Yaskawa INFORM job: A_ROOF_SIDE_0617_2_PAINT_15.JBI

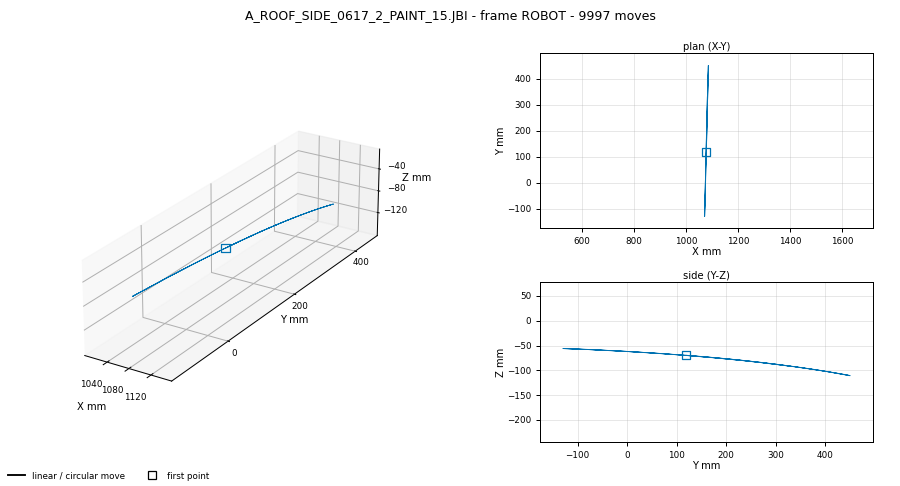
[picture p0: tool path of A_ROOF_SIDE_0617_2_PAINT_15.JBI in frame ROBOT, 9997 of 9997 moves have a stored position in this frame; points joined in program order, loops and branches not executed]
/JOB
//NAME A_ROOF_SIDE_0617_2_PAINT15
//POS
///NPOS 9997,0,0,0,0,0
///TOOL 1
///USER 0
///POSTYPE ROBOT
///RECTAN
///RCONF 1,0,0,0,0,0,0,0,0,0,0,0,0,0,0,0,0,0,0,0,0,0,0,0
C00000=1077.480,118.729,-69.527,173.974,23.685,154.115
C00001=1077.485,118.978,-69.546,173.976,23.687,154.116
C00002=1077.491,119.227,-69.566,173.978,23.689,154.116
C00003=1077.497,119.476,-69.585,173.979,23.692,154.116
C00004=1077.502,119.725,-69.604,173.982,23.695,154.116
C00005=1077.508,119.975,-69.623,173.983,23.697,154.117
C00006=1077.514,120.224,-69.643,173.984,23.699,154.117
C00007=1077.520,120.473,-69.663,173.987,23.702,154.117
C00008=1077.525,120.722,-69.682,173.988,23.704,154.117
C00009=1077.531,120.971,-69.702,173.990,23.707,154.118
C00010=1077.537,121.220,-69.721,173.991,23.709,154.118
C00011=1077.542,121.470,-69.740,173.994,23.711,154.118
C00012=1077.547,121.719,-69.761,173.995,23.714,154.118
C00013=1077.553,121.968,-69.780,173.997,23.716,154.119
C00014=1077.559,122.218,-69.799,173.999,23.719,154.119
C00015=1077.565,122.466,-69.819,174.001,23.721,154.119
C00016=1077.570,122.715,-69.838,174.002,23.723,154.119
C00017=1077.576,122.965,-69.857,174.004,23.726,154.120
C00018=1077.582,123.213,-69.877,174.006,23.728,154.120
C00019=1077.587,123.463,-69.896,174.007,23.730,154.120
C00020=1077.593,123.712,-69.916,174.010,23.733,154.120
C00021=1077.598,123.961,-69.936,174.011,23.735,154.121
C00022=1077.604,124.211,-69.955,174.013,23.738,154.121
C00023=1077.610,124.460,-69.975,174.015,23.740,154.121
C00024=1077.616,124.709,-69.995,174.017,23.743,154.121
C00025=1077.622,124.958,-70.015,174.018,23.745,154.122
C00026=1077.627,125.207,-70.034,174.021,23.747,154.122
C00027=1077.633,125.456,-70.054,174.022,23.750,154.122
C00028=1077.638,125.706,-70.074,174.024,23.752,154.122
C00029=1077.644,125.955,-70.094,174.026,23.754,154.123
C00030=1077.650,126.204,-70.113,174.028,23.757,154.123
C00031=1077.656,126.453,-70.133,174.029,23.759,154.123
C00032=1077.662,126.702,-70.152,174.031,23.761,154.123
C00033=1077.668,126.983,-70.174,174.033,23.764,154.124
C00034=1077.674,127.265,-70.197,174.035,23.767,154.124
C00035=1077.681,127.545,-70.219,174.037,23.769,154.124
C00036=1077.687,127.826,-70.242,174.039,23.772,154.124
C00037=1077.693,128.075,-70.261,174.041,23.775,154.125
C00038=1077.699,128.324,-70.281,174.043,23.777,154.125
C00039=1077.704,128.574,-70.301,174.045,23.779,154.125
C00040=1077.710,128.823,-70.321,174.047,23.782,154.125
C00041=1077.716,129.072,-70.340,174.048,23.784,154.125
C00042=1077.722,129.321,-70.360,174.050,23.786,154.126
C00043=1077.728,129.570,-70.380,174.052,23.789,154.126
C00044=1077.733,129.819,-70.400,174.054,23.791,154.126
C00045=1077.739,130.068,-70.420,174.056,23.793,154.126
C00046=1077.745,130.317,-70.439,174.058,23.796,154.127
C00047=1077.750,130.567,-70.459,174.059,23.798,154.127
C00048=1077.756,130.815,-70.479,174.062,23.800,154.127
C00049=1077.762,131.065,-70.500,174.063,23.803,154.127
C00050=1077.768,131.315,-70.519,174.065,23.805,154.128
C00051=1077.774,131.563,-70.539,174.067,23.807,154.128
C00052=1077.780,131.812,-70.559,174.069,23.810,154.128
C00053=1077.785,132.062,-70.579,174.070,23.812,154.128
C00054=1077.791,132.311,-70.599,174.073,23.814,154.128
C00055=1077.797,132.560,-70.619,174.074,23.817,154.129
C00056=1077.802,132.809,-70.639,174.076,23.819,154.129
C00057=1077.808,133.058,-70.658,174.078,23.821,154.129
C00058=1077.813,133.307,-70.679,174.080,23.824,154.129
C00059=1077.819,133.556,-70.699,174.081,23.826,154.130
C00060=1077.824,133.805,-70.719,174.084,23.829,154.130
C00061=1077.830,134.055,-70.739,174.085,23.831,154.130
C00062=1077.835,134.304,-70.759,174.087,23.833,154.130
C00063=1077.841,134.553,-70.779,174.089,23.836,154.131
C00064=1077.846,134.802,-70.800,174.091,23.838,154.131
C00065=1077.853,135.051,-70.820,174.092,23.840,154.131
C00066=1077.859,135.300,-70.840,174.095,23.843,154.131
C00067=1077.864,135.550,-70.860,174.096,23.845,154.132
C00068=1077.870,135.799,-70.880,174.098,23.848,154.132
C00069=1077.875,136.048,-70.900,174.100,23.850,154.132
C00070=1077.881,136.297,-70.920,174.102,23.853,154.132
C00071=1077.886,136.546,-70.941,174.103,23.854,154.132
C00072=1077.892,136.794,-70.961,174.106,23.857,154.133
C00073=1077.898,137.044,-70.981,174.108,23.859,154.133
C00074=1077.904,137.293,-71.002,174.109,23.862,154.133
C00075=1077.910,137.542,-71.022,174.112,23.864,154.133
C00076=1077.915,137.792,-71.041,174.113,23.866,154.133
C00077=1077.920,138.041,-71.062,174.115,23.869,154.134
C00078=1077.926,138.290,-71.082,174.117,23.871,154.134
C00079=1077.932,138.539,-71.103,174.119,23.874,154.134
C00080=1077.937,138.788,-71.123,174.120,23.876,154.134
C00081=1077.944,139.037,-71.143,174.123,23.878,154.135
C00082=1077.949,139.286,-71.164,174.124,23.881,154.135
C00083=1077.955,139.535,-71.184,174.126,23.883,154.135
C00084=1077.960,139.784,-71.204,174.128,23.885,154.135
C00085=1077.966,140.033,-71.224,174.130,23.888,154.136
C00086=1077.971,140.282,-71.245,174.132,23.890,154.136
C00087=1077.977,140.532,-71.266,174.134,23.892,154.136
C00088=1077.983,140.781,-71.286,174.136,23.895,154.136
C00089=1077.988,141.030,-71.306,174.137,23.897,154.136
C00090=1077.994,141.279,-71.327,174.140,23.900,154.137
C00091=1078.000,141.527,-71.348,174.141,23.902,154.137
C00092=1078.005,141.777,-71.368,174.143,23.904,154.137
C00093=1078.010,142.026,-71.389,174.145,23.907,154.137
C00094=1078.016,142.276,-71.410,174.147,23.909,154.138
C00095=1078.022,142.524,-71.430,174.149,23.912,154.138
C00096=1078.028,142.773,-71.450,174.151,23.913,154.138
C00097=1078.034,143.054,-71.473,174.153,23.916,154.138
C00098=1078.040,143.335,-71.497,174.155,23.919,154.139
C00099=1078.047,143.616,-71.520,174.158,23.922,154.139
C00100=1078.053,143.897,-71.543,174.160,23.924,154.139
C00101=1078.058,144.146,-71.563,174.161,23.927,154.139
C00102=1078.064,144.395,-71.585,174.164,23.929,154.139
C00103=1078.071,144.644,-71.605,174.166,23.932,154.140
C00104=1078.076,144.893,-71.625,174.167,23.933,154.140
C00105=1078.081,145.143,-71.646,174.170,23.936,154.140
C00106=1078.086,145.392,-71.667,174.171,23.938,154.140
C00107=1078.093,145.641,-71.688,174.173,23.941,154.141
C00108=1078.098,145.890,-71.708,174.175,23.943,154.141
C00109=1078.104,146.139,-71.729,174.177,23.945,154.141
C00110=1078.109,146.388,-71.749,174.179,23.948,154.141
C00111=1078.116,146.637,-71.770,174.181,23.950,154.141
C00112=1078.121,146.886,-71.791,174.183,23.953,154.142
C00113=1078.126,147.135,-71.811,174.185,23.954,154.142
C00114=1078.133,147.384,-71.833,174.187,23.957,154.142
C00115=1078.138,147.633,-71.854,174.189,23.959,154.142
C00116=1078.144,147.882,-71.874,174.190,23.962,154.143
C00117=1078.149,148.131,-71.894,174.193,23.964,154.143
C00118=1078.155,148.381,-71.916,174.194,23.966,154.143
C00119=1078.160,148.630,-71.936,174.196,23.969,154.143
C00120=1078.166,148.878,-71.958,174.199,23.971,154.143
C00121=1078.172,149.128,-71.979,174.200,23.973,154.144
C00122=1078.177,149.377,-71.999,174.203,23.976,154.144
C00123=1078.183,149.625,-72.020,174.204,23.978,154.144
C00124=1078.189,149.874,-72.040,174.206,23.981,154.144
C00125=1078.195,150.124,-72.061,174.209,23.983,154.145
C00126=1078.200,150.373,-72.082,174.210,23.985,154.145
C00127=1078.205,150.622,-72.103,174.212,23.987,154.145
C00128=1078.212,150.871,-72.125,174.214,23.990,154.145
C00129=1078.217,151.120,-72.145,174.216,23.992,154.145
C00130=1078.222,151.369,-72.166,174.218,23.995,154.146
C00131=1078.228,151.619,-72.187,174.220,23.997,154.146
C00132=1078.234,151.867,-72.209,174.222,23.999,154.146
C00133=1078.239,152.116,-72.229,174.224,24.002,154.146
C00134=1078.245,152.365,-72.251,174.226,24.004,154.147
C00135=1078.250,152.614,-72.271,174.228,24.007,154.147
C00136=1078.256,152.863,-72.293,174.230,24.008,154.147
C00137=1078.262,153.113,-72.314,174.232,24.011,154.147
C00138=1078.267,153.361,-72.335,174.234,24.013,154.147
C00139=1078.273,153.610,-72.355,174.236,24.016,154.148
C00140=1078.279,153.860,-72.377,174.238,24.018,154.148
C00141=1078.284,154.109,-72.398,174.240,24.021,154.148
C00142=1078.290,154.358,-72.419,174.242,24.022,154.148
C00143=1078.296,154.607,-72.440,174.244,24.025,154.149
C00144=1078.301,154.856,-72.461,174.245,24.027,154.149
C00145=1078.307,155.105,-72.483,174.248,24.030,154.149
C00146=1078.312,155.354,-72.503,174.250,24.032,154.149
C00147=1078.319,155.603,-72.525,174.251,24.034,154.149
C00148=1078.324,155.852,-72.546,174.254,24.036,154.150
C00149=1078.329,156.101,-72.567,174.256,24.039,154.150
C00150=1078.335,156.350,-72.589,174.257,24.041,154.150
C00151=1078.340,156.599,-72.610,174.260,24.044,154.150
C00152=1078.346,156.848,-72.631,174.262,24.046,154.150
C00153=1078.352,157.097,-72.652,174.264,24.048,154.151
C00154=1078.357,157.346,-72.674,174.266,24.051,154.151
C00155=1078.363,157.595,-72.695,174.268,24.053,154.151
C00156=1078.368,157.844,-72.716,174.270,24.055,154.151
C00157=1078.374,158.093,-72.738,174.272,24.058,154.151
C00158=1078.380,158.343,-72.759,174.274,24.060,154.152
C00159=1078.385,158.591,-72.780,174.276,24.062,154.152
C00160=1078.391,158.840,-72.802,174.278,24.065,154.152
C00161=1078.398,159.121,-72.825,174.280,24.068,154.152
C00162=1078.404,159.402,-72.850,174.283,24.070,154.153
C00163=1078.410,159.682,-72.874,174.285,24.072,154.153
C00164=1078.417,159.963,-72.898,174.287,24.075,154.153
C00165=1078.422,160.212,-72.919,174.290,24.077,154.153
C00166=1078.427,160.461,-72.941,174.291,24.080,154.154
C00167=1078.433,160.710,-72.963,174.293,24.082,154.154
C00168=1078.439,160.959,-72.983,174.296,24.085,154.154
C00169=1078.445,161.208,-73.005,174.297,24.086,154.154
C00170=1078.450,161.457,-73.026,174.299,24.089,154.154
C00171=1078.456,161.706,-73.048,174.302,24.091,154.155
C00172=1078.461,161.955,-73.070,174.303,24.094,154.155
C00173=1078.467,162.204,-73.092,174.305,24.096,154.155
C00174=1078.472,162.453,-73.113,174.308,24.099,154.155
C00175=1078.478,162.702,-73.135,174.310,24.101,154.155
C00176=1078.483,162.951,-73.157,174.311,24.104,154.156
C00177=1078.488,163.200,-73.178,174.314,24.106,154.156
C00178=1078.494,163.449,-73.199,174.316,24.109,154.156
C00179=1078.499,163.698,-73.221,174.317,24.111,154.156
C00180=1078.505,163.947,-73.243,174.320,24.113,154.157
C00181=1078.510,164.196,-73.265,174.322,24.116,154.157
C00182=1078.516,164.446,-73.286,174.324,24.118,154.157
C00183=1078.521,164.694,-73.308,174.326,24.120,154.157
C00184=1078.527,164.944,-73.330,174.328,24.123,154.158
C00185=1078.532,165.192,-73.352,174.330,24.125,154.158
C00186=1078.538,165.442,-73.373,174.332,24.128,154.158
C00187=1078.543,165.690,-73.395,174.334,24.130,154.158
C00188=1078.549,165.940,-73.417,174.336,24.132,154.158
C00189=1078.554,166.188,-73.439,174.338,24.134,154.159
C00190=1078.560,166.437,-73.461,174.340,24.137,154.159
C00191=1078.565,166.686,-73.483,174.343,24.140,154.159
C00192=1078.571,166.935,-73.505,174.345,24.142,154.159
C00193=1078.576,167.184,-73.526,174.346,24.144,154.160
C00194=1078.582,167.433,-73.548,174.349,24.146,154.160
C00195=1078.587,167.682,-73.570,174.351,24.149,154.160
C00196=1078.592,167.931,-73.592,174.352,24.151,154.160
C00197=1078.598,168.180,-73.613,174.355,24.154,154.160
C00198=1078.603,168.429,-73.636,174.357,24.156,154.161
C00199=1078.609,168.677,-73.658,174.359,24.159,154.161
C00200=1078.615,168.927,-73.680,174.361,24.161,154.161
C00201=1078.620,169.175,-73.701,174.363,24.163,154.161
C00202=1078.626,169.425,-73.723,174.365,24.166,154.161
C00203=1078.632,169.674,-73.745,174.368,24.168,154.162
C00204=1078.637,169.923,-73.767,174.369,24.170,154.162
C00205=1078.642,170.172,-73.790,174.372,24.172,154.162
C00206=1078.648,170.420,-73.811,174.374,24.175,154.162
C00207=1078.653,170.670,-73.833,174.376,24.177,154.162
C00208=1078.660,170.919,-73.855,174.378,24.180,154.163
C00209=1078.665,171.167,-73.878,174.380,24.182,154.163
C00210=1078.670,171.417,-73.900,174.382,24.185,154.163
C00211=1078.676,171.665,-73.921,174.385,24.187,154.163
C00212=1078.681,171.915,-73.943,174.386,24.189,154.164
C00213=1078.688,172.163,-73.966,174.388,24.191,154.164
C00214=1078.692,172.412,-73.987,174.391,24.194,154.164
C00215=1078.698,172.662,-74.010,174.393,24.196,154.164
C00216=1078.704,172.910,-74.032,174.395,24.199,154.164
C00217=1078.709,173.159,-74.054,174.397,24.201,154.165
C00218=1078.715,173.409,-74.076,174.399,24.203,154.165
C00219=1078.721,173.657,-74.099,174.402,24.206,154.165
C00220=1078.726,173.906,-74.120,174.403,24.208,154.165
C00221=1078.732,174.155,-74.142,174.405,24.210,154.165
C00222=1078.738,174.404,-74.165,174.408,24.212,154.166
C00223=1078.743,174.653,-74.187,174.410,24.215,154.166
C00224=1078.749,174.901,-74.209,174.412,24.217,154.166
C00225=1078.755,175.182,-74.235,174.415,24.220,154.166
C00226=1078.761,175.462,-74.260,174.417,24.223,154.166
C00227=1078.768,175.743,-74.284,174.419,24.225,154.167
C00228=1078.774,176.023,-74.309,174.422,24.227,154.167
C00229=1078.780,176.272,-74.332,174.424,24.230,154.167
C00230=1078.785,176.522,-74.354,174.426,24.232,154.167
C00231=1078.791,176.770,-74.376,174.428,24.235,154.168
C00232=1078.796,177.019,-74.398,174.430,24.237,154.168
C00233=1078.802,177.268,-74.421,174.433,24.239,154.168
C00234=1078.809,177.517,-74.443,174.435,24.242,154.168
C00235=1078.813,177.765,-74.465,174.437,24.244,154.168
C00236=1078.819,178.014,-74.488,174.439,24.246,154.169
C00237=1078.825,178.263,-74.510,174.441,24.248,154.169
C00238=1078.831,178.512,-74.533,174.443,24.251,154.169
C00239=1078.837,178.762,-74.555,174.446,24.253,154.169
C00240=1078.842,179.010,-74.578,174.448,24.255,154.169
C00241=1078.848,179.259,-74.599,174.450,24.258,154.170
C00242=1078.854,179.508,-74.622,174.452,24.260,154.170
C00243=1078.859,179.757,-74.645,174.454,24.262,154.170
C00244=1078.865,180.006,-74.667,174.457,24.265,154.170
C00245=1078.871,180.254,-74.689,174.459,24.267,154.170
C00246=1078.876,180.503,-74.712,174.461,24.270,154.171
C00247=1078.882,180.753,-74.735,174.463,24.272,154.171
C00248=1078.888,181.001,-74.757,174.465,24.274,154.171
C00249=1078.894,181.250,-74.780,174.467,24.276,154.171
C00250=1078.899,181.500,-74.802,174.470,24.279,154.171
C00251=1078.905,181.749,-74.825,174.472,24.281,154.171
C00252=1078.911,181.997,-74.847,174.475,24.283,154.172
C00253=1078.916,182.246,-74.869,174.476,24.285,154.172
C00254=1078.922,182.495,-74.892,174.479,24.287,154.172
C00255=1078.928,182.744,-74.915,174.481,24.290,154.172
C00256=1078.934,182.993,-74.938,174.483,24.292,154.172
C00257=1078.940,183.242,-74.960,174.486,24.294,154.173
C00258=1078.945,183.491,-74.983,174.488,24.297,154.173
C00259=1078.951,183.740,-75.006,174.490,24.299,154.173
C00260=1078.957,183.989,-75.029,174.492,24.301,154.173
C00261=1078.963,184.238,-75.050,174.494,24.304,154.173
C00262=1078.968,184.486,-75.073,174.497,24.306,154.173
C00263=1078.974,184.735,-75.096,174.499,24.308,154.174
C00264=1078.980,184.984,-75.119,174.501,24.311,154.174
C00265=1078.985,185.233,-75.142,174.504,24.313,154.174
C00266=1078.991,185.482,-75.165,174.506,24.316,154.174
C00267=1078.997,185.731,-75.187,174.507,24.318,154.174
C00268=1079.002,185.980,-75.210,174.510,24.320,154.175
C00269=1079.007,186.229,-75.233,174.512,24.323,154.175
C00270=1079.012,186.478,-75.256,174.514,24.325,154.175
C00271=1079.018,186.726,-75.279,174.517,24.328,154.175
C00272=1079.024,186.975,-75.302,174.519,24.330,154.176
C00273=1079.030,187.224,-75.325,174.521,24.333,154.176
C00274=1079.035,187.473,-75.348,174.523,24.334,154.176
C00275=1079.040,187.722,-75.371,174.525,24.337,154.176
C00276=1079.045,187.971,-75.394,174.527,24.340,154.177
C00277=1079.051,188.219,-75.417,174.530,24.342,154.177
C00278=1079.057,188.468,-75.440,174.532,24.345,154.177
C00279=1079.062,188.718,-75.463,174.535,24.347,154.177
C00280=1079.068,188.966,-75.486,174.537,24.350,154.177
C00281=1079.073,189.215,-75.509,174.539,24.352,154.177
C00282=1079.079,189.464,-75.532,174.542,24.354,154.178
C00283=1079.084,189.712,-75.555,174.543,24.356,154.178
C00284=1079.089,189.962,-75.578,174.545,24.359,154.178
C00285=1079.095,190.211,-75.601,174.548,24.361,154.178
C00286=1079.101,190.459,-75.624,174.550,24.364,154.179
C00287=1079.106,190.708,-75.647,174.553,24.366,154.179
C00288=1079.111,190.958,-75.671,174.555,24.369,154.179
C00289=1079.118,191.238,-75.697,174.557,24.371,154.179
C00290=1079.124,191.517,-75.722,174.560,24.374,154.180
C00291=1079.131,191.797,-75.749,174.563,24.377,154.180
C00292=1079.136,192.077,-75.775,174.565,24.379,154.180
C00293=1079.142,192.326,-75.798,174.567,24.382,154.180
C00294=1079.148,192.575,-75.821,174.570,24.384,154.180
C00295=1079.153,192.824,-75.844,174.572,24.387,154.181
C00296=1079.159,193.072,-75.868,174.574,24.389,154.181
C00297=1079.165,193.321,-75.891,174.577,24.392,154.181
C00298=1079.170,193.570,-75.914,174.579,24.394,154.181
C00299=1079.175,193.819,-75.937,174.581,24.396,154.181
C00300=1079.181,194.068,-75.960,174.583,24.398,154.182
C00301=1079.187,194.316,-75.984,174.585,24.401,154.182
C00302=1079.192,194.566,-76.008,174.588,24.403,154.182
C00303=1079.198,194.814,-76.031,174.590,24.406,154.182
C00304=1079.204,195.063,-76.054,174.592,24.408,154.182
C00305=1079.210,195.312,-76.077,174.595,24.411,154.183
C00306=1079.215,195.561,-76.101,174.597,24.413,154.183
C00307=1079.221,195.810,-76.124,174.599,24.416,154.183
C00308=1079.227,196.059,-76.148,174.602,24.418,154.183
C00309=1079.232,196.308,-76.171,174.604,24.420,154.184
C00310=1079.238,196.557,-76.194,174.606,24.423,154.184
C00311=1079.244,196.805,-76.218,174.609,24.425,154.184
C00312=1079.249,197.054,-76.241,174.611,24.427,154.184
C00313=1079.255,197.303,-76.264,174.614,24.430,154.184
C00314=1079.261,197.552,-76.288,174.616,24.432,154.184
C00315=1079.266,197.801,-76.312,174.618,24.434,154.185
C00316=1079.272,198.049,-76.335,174.621,24.437,154.185
C00317=1079.277,198.298,-76.358,174.623,24.439,154.185
C00318=1079.283,198.547,-76.383,174.625,24.442,154.185
C00319=1079.289,198.796,-76.406,174.628,24.444,154.185
C00320=1079.294,199.045,-76.429,174.630,24.447,154.186
C00321=1079.300,199.294,-76.453,174.632,24.449,154.186
C00322=1079.306,199.542,-76.476,174.635,24.451,154.186
C00323=1079.311,199.791,-76.500,174.637,24.454,154.186
C00324=1079.317,200.040,-76.523,174.640,24.456,154.186
C00325=1079.323,200.289,-76.547,174.642,24.459,154.187
C00326=1079.328,200.538,-76.571,174.643,24.460,154.187
C00327=1079.334,200.786,-76.594,174.646,24.463,154.187
C00328=1079.339,201.036,-76.618,174.648,24.465,154.187
C00329=1079.345,201.284,-76.641,174.651,24.467,154.187
C00330=1079.351,201.532,-76.665,174.653,24.470,154.188
C00331=1079.357,201.782,-76.689,174.655,24.472,154.188
C00332=1079.363,202.030,-76.713,174.658,24.475,154.188
C00333=1079.368,202.280,-76.736,174.660,24.477,154.188
C00334=1079.374,202.528,-76.760,174.662,24.480,154.189
C00335=1079.380,202.777,-76.785,174.665,24.482,154.189
C00336=1079.386,203.026,-76.807,174.668,24.485,154.189
C00337=1079.391,203.275,-76.832,174.670,24.487,154.189
C00338=1079.396,203.523,-76.856,174.673,24.490,154.189
C00339=1079.402,203.772,-76.879,174.675,24.492,154.189
C00340=1079.407,204.021,-76.903,174.677,24.495,154.190
C00341=1079.413,204.269,-76.927,174.680,24.497,154.190
C00342=1079.419,204.519,-76.951,174.682,24.499,154.190
C00343=1079.424,204.767,-76.975,174.684,24.502,154.190
C00344=1079.430,205.016,-76.999,174.687,24.504,154.191
C00345=1079.435,205.265,-77.022,174.689,24.507,154.191
C00346=1079.441,205.514,-77.046,174.692,24.509,154.191
C00347=1079.447,205.763,-77.071,174.694,24.512,154.191
C00348=1079.453,206.011,-77.095,174.696,24.514,154.191
C00349=1079.458,206.260,-77.119,174.699,24.517,154.192
C00350=1079.463,206.509,-77.143,174.701,24.519,154.192
C00351=1079.470,206.758,-77.167,174.703,24.521,154.192
C00352=1079.475,207.006,-77.191,174.706,24.524,154.192
C00353=1079.498,208.041,-77.291,174.808,24.578,154.191
C00354=1079.507,208.442,-77.330,174.812,24.584,154.192
C00355=1079.516,208.843,-77.371,174.815,24.589,154.192
C00356=1079.526,209.243,-77.410,174.819,24.595,154.193
C00357=1079.535,209.644,-77.449,174.823,24.601,154.194
C00358=1079.541,209.893,-77.474,174.825,24.604,154.194
C00359=1079.546,210.141,-77.499,174.827,24.607,154.194
C00360=1079.552,210.391,-77.523,174.829,24.611,154.195
C00361=1079.558,210.639,-77.548,174.832,24.614,154.195
C00362=1079.564,210.888,-77.573,174.834,24.617,154.196
C00363=1079.569,211.137,-77.597,174.837,24.621,154.196
C00364=1079.575,211.385,-77.622,174.839,24.625,154.197
C00365=1079.580,211.634,-77.647,174.841,24.628,154.197
C00366=1079.586,211.883,-77.673,174.843,24.631,154.198
C00367=1079.592,212.132,-77.697,174.845,24.635,154.198
C00368=1079.598,212.380,-77.722,174.848,24.638,154.198
C00369=1079.603,212.629,-77.747,174.850,24.641,154.199
C00370=1079.609,212.877,-77.772,174.853,24.645,154.199
C00371=1079.615,213.127,-77.796,174.855,24.648,154.200
C00372=1079.621,213.375,-77.821,174.857,24.651,154.200
C00373=1079.626,213.624,-77.846,174.860,24.655,154.201
C00374=1079.631,213.872,-77.872,174.862,24.659,154.201
C00375=1079.637,214.121,-77.896,174.864,24.662,154.201
C00376=1079.643,214.369,-77.921,174.866,24.665,154.202
C00377=1079.649,214.619,-77.946,174.868,24.669,154.202
C00378=1079.654,214.868,-77.972,174.871,24.672,154.203
C00379=1079.659,215.116,-77.996,174.873,24.675,154.203
C00380=1079.666,215.365,-78.021,174.875,24.679,154.204
C00381=1079.671,215.613,-78.046,174.877,24.682,154.204
C00382=1079.677,215.862,-78.071,174.880,24.686,154.204
C00383=1079.683,216.111,-78.097,174.882,24.690,154.205
C00384=1079.688,216.359,-78.122,174.885,24.693,154.205
C00385=1079.694,216.608,-78.146,174.887,24.696,154.206
C00386=1079.700,216.856,-78.171,174.889,24.699,154.206
C00387=1079.705,217.105,-78.197,174.892,24.703,154.207
C00388=1079.711,217.355,-78.222,174.894,24.706,154.207
C00389=1079.717,217.603,-78.247,174.896,24.710,154.208
C00390=1079.722,217.852,-78.273,174.898,24.713,154.208
C00391=1079.728,218.101,-78.297,174.900,24.716,154.208
C00392=1079.734,218.349,-78.322,174.903,24.720,154.209
C00393=1079.740,218.598,-78.348,174.906,24.723,154.209
C00394=1079.745,218.847,-78.374,174.908,24.727,154.210
C00395=1079.751,219.094,-78.399,174.910,24.730,154.210
C00396=1079.757,219.344,-78.423,174.913,24.734,154.211
C00397=1079.762,219.593,-78.449,174.915,24.737,154.211
C00398=1079.768,219.841,-78.474,174.917,24.740,154.211
C00399=1079.774,220.089,-78.500,174.919,24.744,154.212
C00400=1079.780,220.338,-78.525,174.922,24.747,154.212
C00401=1079.785,220.586,-78.550,174.924,24.750,154.213
C00402=1079.791,220.836,-78.575,174.926,24.754,154.213
C00403=1079.797,221.085,-78.601,174.929,24.757,154.214
C00404=1079.803,221.333,-78.626,174.932,24.761,154.214
C00405=1079.808,221.581,-78.651,174.934,24.764,154.214
C00406=1079.817,221.987,-78.693,174.937,24.769,154.215
C00407=1079.827,222.391,-78.735,174.941,24.775,154.216
C00408=1079.835,222.797,-78.776,174.945,24.781,154.216
C00409=1079.845,223.201,-78.818,174.949,24.786,154.217
C00410=1079.851,223.450,-78.844,174.951,24.790,154.218
C00411=1079.857,223.699,-78.869,174.953,24.793,154.218
C00412=1079.863,223.948,-78.895,174.956,24.797,154.218
C00413=1079.867,224.196,-78.920,174.958,24.800,154.219
C00414=1079.874,224.445,-78.946,174.960,24.803,154.219
C00415=1079.879,224.694,-78.972,174.963,24.807,154.220
C00416=1079.885,224.942,-78.997,174.965,24.811,154.220
C00417=1079.890,225.190,-79.023,174.968,24.814,154.221
C00418=1079.896,225.439,-79.048,174.970,24.817,154.221
C00419=1079.902,225.688,-79.074,174.973,24.820,154.222
C00420=1079.907,225.937,-79.100,174.975,24.824,154.222
C00421=1079.914,226.185,-79.126,174.977,24.827,154.222
C00422=1079.919,226.433,-79.151,174.979,24.830,154.223
C00423=1079.925,226.682,-79.177,174.982,24.835,154.223
C00424=1079.930,226.931,-79.203,174.984,24.838,154.224
C00425=1079.937,227.180,-79.228,174.987,24.841,154.224
C00426=1079.942,227.428,-79.255,174.990,24.844,154.225
C00427=1079.948,227.677,-79.281,174.992,24.848,154.225
C00428=1079.954,227.926,-79.306,174.994,24.851,154.225
C00429=1079.959,228.174,-79.331,174.996,24.854,154.226
C00430=1079.964,228.423,-79.357,174.999,24.858,154.226
C00431=1079.971,228.671,-79.383,175.001,24.862,154.227
C00432=1079.976,228.920,-79.409,175.003,24.865,154.227
C00433=1079.983,229.169,-79.435,175.006,24.868,154.228
C00434=1079.988,229.417,-79.461,175.009,24.871,154.228
C00435=1079.994,229.666,-79.487,175.011,24.875,154.228
C00436=1080.000,229.915,-79.513,175.014,24.879,154.229
C00437=1080.006,230.163,-79.539,175.016,24.882,154.229
C00438=1080.011,230.411,-79.565,175.018,24.885,154.230
C00439=1080.016,230.660,-79.591,175.020,24.889,154.230
C00440=1080.023,230.908,-79.617,175.023,24.892,154.231
C00441=1080.028,231.157,-79.643,175.025,24.895,154.231
C00442=1080.034,231.406,-79.669,175.027,24.899,154.231
C00443=1080.039,231.655,-79.695,175.030,24.903,154.232
C00444=1080.045,231.904,-79.721,175.033,24.906,154.232
C00445=1080.051,232.152,-79.747,175.035,24.909,154.233
C00446=1080.057,232.401,-79.773,175.038,24.913,154.233
C00447=1080.063,232.649,-79.800,175.040,24.916,154.234
C00448=1080.068,232.898,-79.826,175.042,24.919,154.234
C00449=1080.073,233.146,-79.852,175.045,24.923,154.235
C00450=1080.079,233.395,-79.878,175.047,24.926,154.235
C00451=1080.084,233.643,-79.905,175.049,24.930,154.235
C00452=1080.091,233.892,-79.930,175.053,24.933,154.236
C00453=1080.096,234.140,-79.957,175.055,24.937,154.236
C00454=1080.102,234.389,-79.983,175.057,24.940,154.237
C00455=1080.108,234.637,-80.009,175.060,24.943,154.237
C00456=1080.113,234.886,-80.036,175.062,24.947,154.238
C00457=1080.119,235.135,-80.062,175.064,24.950,154.238
C00458=1080.128,235.531,-80.104,175.069,24.956,154.239
C00459=1080.137,235.928,-80.146,175.072,24.961,154.239
C00460=1080.146,236.324,-80.188,175.076,24.967,154.240
C00461=1080.155,236.720,-80.230,175.080,24.973,154.241
C00462=1080.161,236.969,-80.256,175.082,24.976,154.241
C00463=1080.166,237.218,-80.283,175.085,24.979,154.242
C00464=1080.173,237.467,-80.310,175.088,24.983,154.242
C00465=1080.178,237.716,-80.336,175.090,24.986,154.243
C00466=1080.184,237.964,-80.363,175.092,24.989,154.243
C00467=1080.190,238.212,-80.389,175.095,24.993,154.243
C00468=1080.196,238.461,-80.416,175.097,24.996,154.244
C00469=1080.201,238.710,-80.442,175.099,25.000,154.244
C00470=1080.207,238.958,-80.469,175.102,25.003,154.245
C00471=1080.213,239.206,-80.495,175.104,25.007,154.245
C00472=1080.218,239.455,-80.522,175.107,25.010,154.246
C00473=1080.224,239.703,-80.548,175.110,25.013,154.246
C00474=1080.229,239.952,-80.576,175.112,25.017,154.246
C00475=1080.235,240.201,-80.602,175.115,25.021,154.247
C00476=1080.240,240.449,-80.628,175.117,25.024,154.247
C00477=1080.246,240.697,-80.655,175.119,25.027,154.248
C00478=1080.253,240.946,-80.682,175.122,25.031,154.248
C00479=1080.258,241.195,-80.709,175.124,25.034,154.249
C00480=1080.264,241.443,-80.735,175.127,25.037,154.249
C00481=1080.270,241.692,-80.762,175.130,25.041,154.250
C00482=1080.276,241.940,-80.789,175.132,25.044,154.250
C00483=1080.281,242.188,-80.815,175.135,25.048,154.250
C00484=1080.287,242.437,-80.842,175.137,25.051,154.251
C00485=1080.293,242.686,-80.869,175.139,25.055,154.251
C00486=1080.299,242.934,-80.896,175.142,25.058,154.252
C00487=1080.304,243.183,-80.923,175.144,25.061,154.252
C00488=1080.310,243.431,-80.949,175.147,25.065,154.253
C00489=1080.315,243.680,-80.977,175.150,25.069,154.253
C00490=1080.321,243.928,-81.003,175.152,25.072,154.253
C00491=1080.327,244.176,-81.030,175.155,25.076,154.254
C00492=1080.332,244.425,-81.057,175.157,25.079,154.254
C00493=1080.338,244.674,-81.084,175.160,25.082,154.255
C00494=1080.344,244.923,-81.111,175.162,25.086,154.255
C00495=1080.349,245.171,-81.139,175.164,25.089,154.256
C00496=1080.355,245.419,-81.165,175.167,25.093,154.256
C00497=1080.361,245.667,-81.192,175.169,25.096,154.257
C00498=1080.367,245.917,-81.220,175.173,25.100,154.257
C00499=1080.372,246.165,-81.246,175.175,25.103,154.257
C00500=1080.378,246.413,-81.273,175.177,25.107,154.258
C00501=1080.383,246.661,-81.301,175.180,25.110,154.258
C00502=1080.389,246.910,-81.328,175.182,25.114,154.259
C00503=1080.396,247.159,-81.355,175.185,25.117,154.259
C00504=1080.401,247.408,-81.382,175.187,25.120,154.260
C00505=1080.407,247.655,-81.409,175.189,25.124,154.260
C00506=1080.412,247.904,-81.436,175.192,25.127,154.260
C00507=1080.417,248.152,-81.463,175.195,25.131,154.261
C00508=1080.423,248.400,-81.491,175.198,25.135,154.261
C00509=1080.429,248.649,-81.518,175.200,25.138,154.262
C00510=1080.437,249.039,-81.561,175.204,25.144,154.263
C00511=1080.445,249.429,-81.604,175.208,25.149,154.263
C00512=1080.455,249.819,-81.647,175.211,25.155,154.264
C00513=1080.463,250.208,-81.690,175.216,25.161,154.265
C00514=1080.470,250.458,-81.717,175.218,25.164,154.265
C00515=1080.475,250.706,-81.745,175.221,25.167,154.266
C00516=1080.481,250.954,-81.771,175.223,25.171,154.266
C00517=1080.486,251.202,-81.799,175.226,25.174,154.266
C00518=1080.492,251.451,-81.827,175.229,25.178,154.267
C00519=1080.498,251.699,-81.854,175.231,25.181,154.267
C00520=1080.503,251.948,-81.881,175.234,25.185,154.268
C00521=1080.510,252.196,-81.909,175.236,25.188,154.268
C00522=1080.515,252.445,-81.936,175.239,25.192,154.269
C00523=1080.520,252.693,-81.964,175.241,25.195,154.269
C00524=1080.526,252.941,-81.991,175.244,25.199,154.270
C00525=1080.532,253.190,-82.019,175.246,25.202,154.270
C00526=1080.538,253.438,-82.047,175.249,25.206,154.271
C00527=1080.543,253.686,-82.074,175.252,25.209,154.271
C00528=1080.549,253.935,-82.102,175.254,25.213,154.271
C00529=1080.555,254.184,-82.129,175.257,25.216,154.272
C00530=1080.560,254.432,-82.157,175.259,25.220,154.272
C00531=1080.566,254.680,-82.185,175.262,25.223,154.273
C00532=1080.572,254.929,-82.212,175.264,25.226,154.273
C00533=1080.578,255.177,-82.240,175.267,25.230,154.274
C00534=1080.583,255.426,-82.268,175.270,25.234,154.274
C00535=1080.589,255.674,-82.295,175.273,25.238,154.275
C00536=1080.595,255.923,-82.323,175.275,25.241,154.275
C00537=1080.600,256.171,-82.351,175.278,25.244,154.275
C00538=1080.607,256.419,-82.379,175.280,25.248,154.276
C00539=1080.612,256.668,-82.406,175.283,25.251,154.276
C00540=1080.617,256.916,-82.434,175.285,25.254,154.277
C00541=1080.624,257.164,-82.462,175.288,25.258,154.277
C00542=1080.629,257.412,-82.490,175.290,25.261,154.278
C00543=1080.635,257.662,-82.517,175.293,25.265,154.278
C00544=1080.641,257.909,-82.545,175.296,25.269,154.279
C00545=1080.647,258.158,-82.573,175.298,25.272,154.279
C00546=1080.652,258.406,-82.601,175.301,25.276,154.280
C00547=1080.658,258.655,-82.629,175.303,25.279,154.280
C00548=1080.664,258.903,-82.657,175.306,25.282,154.280
C00549=1080.670,259.151,-82.685,175.308,25.286,154.281
C00550=1080.675,259.400,-82.713,175.311,25.289,154.281
C00551=1080.682,259.649,-82.740,175.314,25.293,154.282
C00552=1080.687,259.897,-82.768,175.317,25.297,154.282
C00553=1080.693,260.145,-82.796,175.319,25.300,154.283
C00554=1080.698,260.393,-82.824,175.322,25.304,154.283
C00555=1080.705,260.642,-82.852,175.325,25.307,154.283
C00556=1080.710,260.890,-82.880,175.327,25.310,154.284
C00557=1080.716,261.139,-82.908,175.330,25.314,154.284
C00558=1080.722,261.387,-82.936,175.332,25.317,154.285
C00559=1080.728,261.636,-82.964,175.336,25.321,154.285
C00560=1080.734,261.884,-82.992,175.338,25.324,154.286
C00561=1080.740,262.132,-83.020,175.341,25.328,154.286
C00562=1080.749,262.519,-83.065,175.344,25.333,154.287
C00563=1080.758,262.906,-83.108,175.349,25.338,154.287
C00564=1080.767,263.293,-83.152,175.353,25.344,154.288
C00565=1080.776,263.680,-83.196,175.357,25.349,154.289
C00566=1080.782,263.928,-83.224,175.360,25.353,154.289
C00567=1080.788,264.177,-83.253,175.363,25.357,154.290
C00568=1080.794,264.425,-83.281,175.365,25.360,154.290
C00569=1080.800,264.674,-83.309,175.368,25.364,154.291
C00570=1080.805,264.921,-83.338,175.370,25.367,154.291
C00571=1080.811,265.170,-83.366,175.373,25.371,154.292
C00572=1080.817,265.418,-83.394,175.375,25.374,154.292
C00573=1080.823,265.667,-83.422,175.378,25.378,154.293
C00574=1080.829,265.915,-83.451,175.381,25.381,154.293
C00575=1080.834,266.163,-83.479,175.384,25.385,154.293
C00576=1080.840,266.412,-83.507,175.387,25.388,154.294
C00577=1080.845,266.660,-83.537,175.389,25.392,154.294
C00578=1080.851,266.908,-83.565,175.392,25.395,154.295
C00579=1080.857,267.157,-83.593,175.394,25.399,154.295
C00580=1080.862,267.404,-83.622,175.397,25.403,154.296
C00581=1080.868,267.653,-83.650,175.399,25.406,154.296
C00582=1080.874,267.902,-83.679,175.402,25.410,154.297
C00583=1080.880,268.149,-83.707,175.405,25.413,154.297
C00584=1080.886,268.398,-83.736,175.408,25.417,154.298
C00585=1080.892,268.646,-83.765,175.411,25.421,154.298
C00586=1080.897,268.895,-83.793,175.413,25.424,154.298
C00587=1080.903,269.143,-83.822,175.416,25.428,154.299
C00588=1080.909,269.392,-83.851,175.418,25.431,154.299
C00589=1080.914,269.640,-83.879,175.421,25.435,154.300
C00590=1080.921,269.888,-83.908,175.423,25.438,154.300
C00591=1080.926,270.137,-83.937,175.426,25.442,154.301
C00592=1080.931,270.384,-83.965,175.429,25.445,154.301
C00593=1080.938,270.632,-83.994,175.432,25.449,154.302
C00594=1080.944,270.881,-84.023,175.435,25.453,154.302
C00595=1080.949,271.129,-84.051,175.437,25.456,154.303
C00596=1080.955,271.378,-84.080,175.440,25.460,154.303
C00597=1080.961,271.626,-84.109,175.442,25.463,154.304
C00598=1080.967,271.874,-84.138,175.445,25.467,154.304
C00599=1080.972,272.122,-84.167,175.448,25.470,154.305
C00600=1080.978,272.370,-84.196,175.451,25.474,154.305
C00601=1080.984,272.619,-84.224,175.454,25.478,154.306
C00602=1080.990,272.867,-84.253,175.456,25.481,154.306
C00603=1080.995,273.115,-84.283,175.459,25.485,154.307
C00604=1081.001,273.364,-84.311,175.462,25.489,154.307
C00605=1081.007,273.612,-84.340,175.464,25.492,154.307
C00606=1081.013,273.860,-84.370,175.467,25.496,154.308
C00607=1081.018,274.108,-84.398,175.469,25.499,154.308
C00608=1081.024,274.357,-84.427,175.472,25.503,154.309
C00609=1081.030,274.605,-84.456,175.475,25.507,154.309
C00610=1081.036,274.853,-84.485,175.478,25.510,154.310
C00611=1081.041,275.101,-84.514,175.481,25.514,154.310
C00612=1081.047,275.349,-84.544,175.483,25.517,154.311
C00613=1081.052,275.598,-84.572,175.486,25.521,154.311
C00614=1081.062,275.988,-84.618,175.491,25.527,154.312
C00615=1081.071,276.378,-84.664,175.494,25.532,154.313
C00616=1081.080,276.768,-84.710,175.499,25.538,154.314
C00617=1081.089,277.157,-84.756,175.503,25.544,154.314
C00618=1081.095,277.406,-84.785,175.505,25.548,154.315
C00619=1081.100,277.654,-84.815,175.509,25.551,154.315
C00620=1081.107,277.902,-84.844,175.512,25.555,154.316
C00621=1081.112,278.151,-84.873,175.514,25.559,154.316
C00622=1081.118,278.399,-84.902,175.517,25.562,154.317
C00623=1081.123,278.647,-84.931,175.519,25.566,154.317
C00624=1081.129,278.895,-84.961,175.522,25.570,154.318
C00625=1081.135,279.143,-84.991,175.525,25.573,154.318
C00626=1081.141,279.391,-85.020,175.527,25.577,154.319
C00627=1081.147,279.640,-85.049,175.530,25.581,154.319
C00628=1081.152,279.888,-85.079,175.534,25.584,154.320
C00629=1081.158,280.136,-85.108,175.536,25.588,154.320
C00630=1081.164,280.385,-85.138,175.539,25.592,154.321
C00631=1081.170,280.633,-85.167,175.542,25.595,154.321
C00632=1081.175,280.881,-85.196,175.544,25.599,154.321
C00633=1081.181,281.129,-85.225,175.547,25.603,154.322
C00634=1081.187,281.377,-85.254,175.550,25.606,154.323
C00635=1081.193,281.625,-85.285,175.552,25.610,154.323
C00636=1081.198,281.873,-85.314,175.555,25.613,154.323
C00637=1081.204,282.122,-85.344,175.558,25.617,154.324
C00638=1081.210,282.370,-85.373,175.560,25.621,154.325
C00639=1081.216,282.618,-85.403,175.564,25.624,154.325
C00640=1081.221,282.866,-85.433,175.567,25.628,154.325
C00641=1081.228,283.114,-85.462,175.569,25.632,154.326
C00642=1081.233,283.363,-85.492,175.572,25.636,154.326
C00643=1081.239,283.611,-85.522,175.575,25.640,154.327
C00644=1081.244,283.858,-85.551,175.577,25.643,154.327
C00645=1081.249,284.107,-85.581,175.580,25.647,154.328
C00646=1081.256,284.354,-85.611,175.583,25.651,154.328
C00647=1081.261,284.603,-85.640,175.585,25.654,154.329
C00648=1081.267,284.851,-85.670,175.588,25.658,154.330
C00649=1081.273,285.099,-85.700,175.592,25.662,154.330
C00650=1081.278,285.347,-85.730,175.594,25.665,154.330
C00651=1081.285,285.595,-85.760,175.597,25.669,154.331
C00652=1081.290,285.843,-85.789,175.600,25.673,154.331
C00653=1081.296,286.092,-85.819,175.602,25.677,154.332
C00654=1081.302,286.340,-85.849,175.605,25.680,154.332
C00655=1081.307,286.588,-85.879,175.608,25.684,154.333
C00656=1081.314,286.836,-85.909,175.610,25.688,154.333
C00657=1081.320,287.085,-85.939,175.613,25.692,154.334
C00658=1081.326,287.333,-85.969,175.616,25.696,154.335
C00659=1081.331,287.581,-85.999,175.620,25.699,154.335
C00660=1081.337,287.829,-86.029,175.622,25.703,154.335
C00661=1081.343,288.077,-86.060,175.625,25.707,154.336
C00662=1081.348,288.325,-86.089,175.628,25.710,154.336
C00663=1081.355,288.573,-86.119,175.630,25.714,154.337
C00664=1081.360,288.821,-86.149,175.633,25.717,154.337
C00665=1081.366,289.069,-86.179,175.636,25.721,154.338
C00666=1081.376,289.469,-86.228,175.641,25.728,154.339
C00667=1081.384,289.869,-86.276,175.645,25.734,154.340
C00668=1081.394,290.269,-86.325,175.650,25.740,154.340
C00669=1081.404,290.668,-86.373,175.654,25.746,154.341
C00670=1081.409,290.916,-86.404,175.656,25.749,154.342
C00671=1081.415,291.164,-86.434,175.659,25.753,154.342
C00672=1081.421,291.412,-86.464,175.663,25.757,154.343
C00673=1081.426,291.660,-86.494,175.666,25.761,154.343
C00674=1081.433,291.909,-86.525,175.668,25.765,154.344
C00675=1081.439,292.156,-86.555,175.671,25.768,154.344
C00676=1081.444,292.405,-86.586,175.674,25.772,154.345
C00677=1081.449,292.653,-86.616,175.677,25.776,154.345
C00678=1081.455,292.901,-86.646,175.679,25.780,154.346
C00679=1081.461,293.149,-86.676,175.682,25.784,154.346
C00680=1081.467,293.397,-86.707,175.685,25.787,154.347
C00681=1081.473,293.645,-86.737,175.688,25.791,154.347
C00682=1081.479,293.893,-86.768,175.691,25.795,154.348
C00683=1081.485,294.141,-86.798,175.694,25.799,154.349
C00684=1081.490,294.389,-86.829,175.697,25.803,154.349
C00685=1081.496,294.637,-86.859,175.700,25.807,154.350
C00686=1081.502,294.885,-86.890,175.702,25.810,154.350
C00687=1081.508,295.133,-86.920,175.705,25.814,154.351
C00688=1081.514,295.381,-86.951,175.708,25.818,154.351
C00689=1081.520,295.629,-86.981,175.711,25.822,154.352
C00690=1081.526,295.877,-87.012,175.713,25.826,154.352
C00691=1081.531,296.125,-87.043,175.716,25.829,154.353
C00692=1081.537,296.373,-87.073,175.719,25.833,154.353
C00693=1081.543,296.621,-87.104,175.722,25.838,154.354
C00694=1081.549,296.869,-87.134,175.725,25.842,154.354
C00695=1081.554,297.118,-87.165,175.727,25.845,154.355
C00696=1081.560,297.365,-87.196,175.731,25.849,154.356
C00697=1081.566,297.613,-87.226,175.734,25.853,154.356
C00698=1081.572,297.861,-87.258,175.737,25.857,154.357
C00699=1081.578,298.109,-87.288,175.740,25.861,154.357
C00700=1081.583,298.357,-87.319,175.742,25.864,154.358
C00701=1081.589,298.605,-87.350,175.745,25.869,154.358
C00702=1081.594,298.853,-87.380,175.748,25.873,154.359
C00703=1081.600,299.101,-87.412,175.751,25.877,154.359
C00704=1081.606,299.349,-87.442,175.753,25.880,154.360
C00705=1081.611,299.597,-87.473,175.756,25.885,154.361
C00706=1081.617,299.845,-87.504,175.759,25.889,154.361
C00707=1081.622,300.093,-87.535,175.762,25.892,154.362
C00708=1081.628,300.341,-87.567,175.765,25.897,154.362
C00709=1081.634,300.589,-87.597,175.767,25.900,154.363
C00710=1081.639,300.837,-87.629,175.770,25.904,154.363
C00711=1081.646,301.085,-87.659,175.774,25.908,154.364
C00712=1081.651,301.333,-87.691,175.776,25.913,154.364
C00713=1081.657,301.581,-87.721,175.780,25.917,154.365
C00714=1081.662,301.829,-87.752,175.783,25.920,154.366
C00715=1081.669,302.077,-87.784,175.785,25.924,154.366
C00716=1081.674,302.325,-87.815,175.788,25.928,154.367
C00717=1081.680,302.572,-87.846,175.791,25.932,154.367
C00718=1081.689,302.987,-87.898,175.795,25.939,154.368
C00719=1081.698,303.401,-87.950,175.801,25.946,154.369
C00720=1081.709,303.815,-88.002,175.805,25.952,154.370
C00721=1081.718,304.229,-88.054,175.810,25.959,154.371
C00722=1081.724,304.476,-88.085,175.814,25.963,154.372
C00723=1081.730,304.725,-88.117,175.816,25.967,154.372
C00724=1081.735,304.973,-88.148,175.819,25.971,154.373
C00725=1081.742,305.220,-88.179,175.822,25.975,154.373
C00726=1081.747,305.469,-88.211,175.825,25.979,154.374
C00727=1081.753,305.716,-88.242,175.828,25.983,154.374
C00728=1081.759,305.964,-88.274,175.831,25.987,154.375
C00729=1081.764,306.212,-88.305,175.834,25.991,154.376
C00730=1081.771,306.460,-88.336,175.836,25.995,154.376
C00731=1081.777,306.708,-88.368,175.839,25.999,154.377
C00732=1081.782,306.955,-88.399,175.842,26.003,154.377
C00733=1081.788,307.204,-88.430,175.845,26.007,154.378
C00734=1081.794,307.451,-88.462,175.848,26.011,154.378
C00735=1081.800,307.700,-88.494,175.851,26.016,154.379
C00736=1081.806,307.947,-88.525,175.854,26.020,154.380
C00737=1081.812,308.196,-88.556,175.857,26.023,154.380
C00738=1081.817,308.443,-88.588,175.859,26.027,154.381
C00739=1081.823,308.691,-88.620,175.863,26.031,154.381
C00740=1081.830,308.939,-88.651,175.866,26.036,154.382
C00741=1081.835,309.187,-88.683,175.869,26.040,154.383
C00742=1081.841,309.435,-88.715,175.872,26.043,154.383
C00743=1081.847,309.682,-88.746,175.875,26.048,154.384
C00744=1081.853,309.931,-88.777,175.878,26.052,154.384
C00745=1081.858,310.178,-88.809,175.881,26.056,154.385
C00746=1081.864,310.427,-88.841,175.884,26.060,154.385
C00747=1081.871,310.675,-88.873,175.886,26.064,154.386
C00748=1081.876,310.922,-88.904,175.889,26.068,154.387
C00749=1081.882,311.170,-88.936,175.892,26.072,154.387
C00750=1081.888,311.418,-88.967,175.895,26.076,154.388
C00751=1081.894,311.666,-88.999,175.898,26.080,154.388
C00752=1081.900,311.914,-89.031,175.901,26.084,154.389
C00753=1081.906,312.161,-89.063,175.904,26.088,154.389
C00754=1081.912,312.410,-89.095,175.907,26.092,154.390
C00755=1081.918,312.658,-89.126,175.910,26.097,154.391
C00756=1081.924,312.905,-89.158,175.914,26.100,154.391
C00757=1081.930,313.153,-89.191,175.916,26.105,154.392
C00758=1081.936,313.401,-89.223,175.919,26.108,154.392
C00759=1081.943,313.649,-89.254,175.922,26.113,154.393
C00760=1081.948,313.896,-89.286,175.925,26.117,154.394
C00761=1081.954,314.145,-89.318,175.928,26.121,154.394
C00762=1081.960,314.393,-89.350,175.931,26.125,154.395
C00763=1081.966,314.641,-89.382,175.934,26.129,154.395
C00764=1081.972,314.888,-89.414,175.937,26.133,154.396
C00765=1081.978,315.136,-89.446,175.940,26.137,154.397
C00766=1081.983,315.384,-89.478,175.943,26.142,154.397
C00767=1081.989,315.632,-89.510,175.946,26.146,154.398
C00768=1081.996,315.879,-89.543,175.949,26.151,154.399
C00769=1082.000,316.127,-89.575,175.952,26.155,154.399
C00770=1082.010,316.545,-89.630,175.956,26.161,154.400
C00771=1082.020,316.961,-89.683,175.962,26.169,154.401
C00772=1082.030,317.379,-89.738,175.967,26.176,154.402
C00773=1082.040,317.796,-89.793,175.971,26.183,154.403
C00774=1082.044,318.043,-89.825,175.974,26.188,154.404
C00775=1082.050,318.292,-89.857,175.977,26.192,154.405
C00776=1082.057,318.539,-89.890,175.980,26.196,154.405
C00777=1082.063,318.787,-89.922,175.983,26.201,154.406
C00778=1082.068,319.035,-89.955,175.986,26.205,154.407
C00779=1082.074,319.283,-89.987,175.989,26.209,154.407
C00780=1082.080,319.530,-90.020,175.992,26.214,154.408
C00781=1082.086,319.779,-90.052,175.995,26.218,154.409
C00782=1082.091,320.026,-90.085,175.998,26.222,154.409
C00783=1082.097,320.274,-90.117,176.001,26.226,154.410
C00784=1082.103,320.522,-90.149,176.004,26.231,154.411
C00785=1082.109,320.770,-90.183,176.007,26.235,154.411
C00786=1082.115,321.018,-90.215,176.010,26.239,154.412
C00787=1082.120,321.265,-90.247,176.013,26.244,154.412
C00788=1082.126,321.513,-90.280,176.016,26.248,154.413
C00789=1082.132,321.761,-90.312,176.019,26.252,154.414
C00790=1082.138,322.008,-90.345,176.022,26.257,154.414
C00791=1082.143,322.257,-90.378,176.025,26.261,154.415
C00792=1082.150,322.505,-90.411,176.029,26.266,154.416
C00793=1082.155,322.751,-90.443,176.032,26.270,154.416
C00794=1082.161,322.999,-90.476,176.035,26.274,154.417
C00795=1082.167,323.248,-90.508,176.038,26.279,154.418
C00796=1082.173,323.495,-90.541,176.041,26.283,154.418
C00797=1082.179,323.743,-90.574,176.044,26.287,154.419
C00798=1082.185,323.991,-90.607,176.047,26.292,154.420
C00799=1082.190,324.239,-90.640,176.050,26.296,154.420
C00800=1082.197,324.487,-90.672,176.052,26.301,154.421
C00801=1082.203,324.734,-90.705,176.055,26.305,154.422
C00802=1082.209,324.982,-90.739,176.058,26.310,154.422
C00803=1082.215,325.230,-90.771,176.062,26.314,154.423
C00804=1082.220,325.478,-90.805,176.065,26.318,154.424
C00805=1082.227,325.725,-90.837,176.068,26.323,154.424
C00806=1082.233,325.973,-90.870,176.071,26.327,154.425
C00807=1082.238,326.221,-90.903,176.074,26.331,154.426
C00808=1082.244,326.469,-90.936,176.077,26.336,154.426
C00809=1082.250,326.717,-90.969,176.080,26.340,154.427
C00810=1082.256,326.965,-91.002,176.083,26.345,154.428
C00811=1082.262,327.212,-91.035,176.086,26.349,154.428
C00812=1082.268,327.460,-91.068,176.089,26.353,154.429
C00813=1082.274,327.708,-91.100,176.092,26.358,154.430
C00814=1082.280,327.955,-91.134,176.095,26.362,154.430
C00815=1082.287,328.202,-91.167,176.098,26.366,154.431
C00816=1082.292,328.450,-91.201,176.101,26.371,154.432
C00817=1082.298,328.698,-91.233,176.104,26.376,154.433
C00818=1082.304,328.946,-91.267,176.108,26.380,154.433
C00819=1082.310,329.193,-91.299,176.111,26.385,154.434
C00820=1082.316,329.441,-91.333,176.114,26.389,154.435
C00821=1082.323,329.690,-91.366,176.116,26.394,154.435
C00822=1082.333,330.100,-91.421,176.122,26.401,154.436
C00823=1082.342,330.510,-91.476,176.126,26.408,154.437
C00824=1082.353,330.921,-91.531,176.131,26.416,154.439
C00825=1082.363,331.331,-91.586,176.137,26.423,154.440
C00826=1082.368,331.578,-91.620,176.140,26.428,154.440
C00827=1082.375,331.826,-91.653,176.143,26.432,154.441
C00828=1082.380,332.074,-91.686,176.146,26.437,154.442
C00829=1082.386,332.321,-91.720,176.149,26.442,154.443
C00830=1082.392,332.570,-91.754,176.152,26.446,154.443
C00831=1082.398,332.818,-91.788,176.156,26.451,154.444
C00832=1082.404,333.065,-91.821,176.159,26.456,154.445
C00833=1082.410,333.313,-91.854,176.162,26.460,154.446
C00834=1082.416,333.560,-91.888,176.165,26.465,154.446
C00835=1082.421,333.808,-91.922,176.168,26.469,154.447
C00836=1082.427,334.055,-91.956,176.170,26.474,154.448
C00837=1082.433,334.304,-91.989,176.173,26.479,154.449
C00838=1082.440,334.551,-92.022,176.176,26.483,154.449
C00839=1082.446,334.799,-92.056,176.179,26.488,154.450
C00840=1082.451,335.046,-92.090,176.183,26.493,154.451
C00841=1082.457,335.294,-92.124,176.186,26.498,154.451
C00842=1082.463,335.542,-92.158,176.189,26.502,154.452
C00843=1082.469,335.790,-92.191,176.192,26.507,154.453
C00844=1082.475,336.037,-92.225,176.195,26.511,154.454
C00845=1082.480,336.285,-92.259,176.198,26.516,154.454
C00846=1082.487,336.532,-92.292,176.202,26.521,154.455
C00847=1082.494,336.780,-92.327,176.205,26.526,154.456
C00848=1082.499,337.028,-92.360,176.208,26.531,154.457
C00849=1082.505,337.275,-92.394,176.211,26.535,154.457
C00850=1082.511,337.523,-92.428,176.214,26.540,154.458
C00851=1082.517,337.770,-92.463,176.217,26.544,154.459
C00852=1082.523,338.018,-92.496,176.220,26.549,154.460
C00853=1082.529,338.265,-92.530,176.224,26.554,154.460
C00854=1082.535,338.513,-92.564,176.227,26.559,154.461
C00855=1082.541,338.761,-92.598,176.230,26.564,154.462
C00856=1082.547,339.009,-92.632,176.232,26.569,154.463
C00857=1082.553,339.257,-92.666,176.235,26.574,154.464
C00858=1082.559,339.504,-92.700,176.239,26.579,154.464
C00859=1082.564,339.751,-92.735,176.242,26.583,154.465
C00860=1082.570,339.999,-92.769,176.245,26.588,154.466
C00861=1082.576,340.247,-92.803,176.248,26.593,154.467
C00862=1082.582,340.494,-92.837,176.251,26.597,154.467
C00863=1082.588,340.741,-92.871,176.255,26.603,154.468
C00864=1082.594,340.989,-92.906,176.258,26.607,154.469
C00865=1082.600,341.237,-92.939,176.261,26.613,154.470
C00866=1082.606,341.484,-92.973,176.264,26.617,154.471
C00867=1082.612,341.733,-93.008,176.267,26.622,154.471
C00868=1082.617,341.980,-93.042,176.271,26.627,154.472
C00869=1082.624,342.227,-93.077,176.274,26.632,154.473
C00870=1082.630,342.475,-93.112,176.277,26.637,154.474
C00871=1082.636,342.722,-93.146,176.279,26.642,154.475
C00872=1082.642,342.970,-93.180,176.283,26.647,154.475
C00873=1082.648,343.218,-93.215,176.286,26.652,154.476
C00874=1082.654,343.466,-93.249,176.289,26.656,154.477
C00875=1082.659,343.714,-93.283,176.292,26.662,154.478
C00876=1082.666,343.962,-93.318,176.296,26.667,154.479
C00877=1082.672,344.211,-93.353,176.299,26.672,154.479
C00878=1082.678,344.459,-93.387,176.302,26.676,154.480
C00879=1082.684,344.706,-93.421,176.305,26.681,154.481
C00880=1082.691,344.953,-93.456,176.309,26.687,154.482
C00881=1082.696,345.201,-93.491,176.312,26.692,154.483
C00882=1082.702,345.449,-93.525,176.315,26.696,154.483
C00883=1082.708,345.696,-93.560,176.317,26.702,154.484
C00884=1082.714,345.943,-93.595,176.321,26.707,154.485
C00885=1082.720,346.191,-93.629,176.324,26.712,154.486
C00886=1082.725,346.439,-93.664,176.327,26.717,154.487
C00887=1082.732,346.686,-93.699,176.330,26.722,154.488
C00888=1082.738,346.933,-93.733,176.334,26.727,154.489
C00889=1082.744,347.182,-93.768,176.337,26.732,154.489
C00890=1082.750,347.428,-93.803,176.340,26.737,154.490
C00891=1082.755,347.677,-93.838,176.344,26.742,154.491
C00892=1082.762,347.923,-93.873,176.346,26.748,154.492
C00893=1082.768,348.171,-93.907,176.349,26.752,154.493
C00894=1082.773,348.418,-93.942,176.352,26.758,154.494
C00895=1082.780,348.666,-93.977,176.356,26.763,154.494
C00896=1082.785,348.913,-94.012,176.359,26.768,154.495
C00897=1082.792,349.161,-94.047,176.362,26.773,154.496
C00898=1082.798,349.409,-94.082,176.366,26.778,154.497
C00899=1082.804,349.656,-94.116,176.369,26.784,154.498
C00900=1082.810,349.904,-94.152,176.372,26.788,154.499
C00901=1082.816,350.151,-94.187,176.375,26.794,154.500
C00902=1082.825,350.555,-94.244,176.381,26.803,154.501
C00903=1082.835,350.959,-94.302,176.386,26.811,154.502
C00904=1082.845,351.363,-94.358,176.391,26.820,154.504
C00905=1082.855,351.767,-94.416,176.396,26.828,154.505
C00906=1082.862,352.014,-94.452,176.399,26.833,154.506
C00907=1082.867,352.262,-94.486,176.403,26.839,154.507
C00908=1082.874,352.509,-94.521,176.406,26.844,154.508
C00909=1082.880,352.757,-94.557,176.409,26.849,154.509
C00910=1082.885,353.004,-94.592,176.412,26.855,154.510
C00911=1082.892,353.251,-94.628,176.415,26.860,154.511
C00912=1082.897,353.499,-94.662,176.418,26.865,154.512
C00913=1082.903,353.747,-94.698,176.422,26.870,154.512
C00914=1082.909,353.994,-94.734,176.425,26.876,154.513
C00915=1082.915,354.241,-94.769,176.428,26.881,154.514
C00916=1082.921,354.489,-94.804,176.432,26.887,154.515
C00917=1082.927,354.736,-94.840,176.435,26.892,154.516
C00918=1082.933,354.984,-94.876,176.437,26.897,154.517
C00919=1082.939,355.231,-94.910,176.441,26.903,154.518
C00920=1082.946,355.478,-94.946,176.444,26.908,154.519
C00921=1082.952,355.726,-94.982,176.448,26.914,154.520
C00922=1082.957,355.973,-95.017,176.451,26.919,154.521
C00923=1082.963,356.221,-95.053,176.454,26.924,154.522
C00924=1082.970,356.468,-95.088,176.458,26.930,154.523
C00925=1082.976,356.716,-95.124,176.460,26.936,154.524
C00926=1082.986,357.122,-95.183,176.466,26.944,154.525
C00927=1082.995,357.531,-95.242,176.472,26.954,154.527
C00928=1083.006,357.939,-95.300,176.477,26.962,154.528
C00929=1083.015,358.347,-95.359,176.482,26.972,154.530
C00930=1083.022,358.594,-95.395,176.486,26.977,154.531
C00931=1083.028,358.841,-95.431,176.488,26.983,154.532
C00932=1083.034,359.088,-95.466,176.492,26.988,154.533
C00933=1083.040,359.335,-95.503,176.495,26.994,154.534
C00934=1083.046,359.583,-95.538,176.498,26.999,154.535
C00935=1083.052,359.831,-95.574,176.502,27.005,154.535
C00936=1083.058,360.078,-95.611,176.505,27.011,154.537
C00937=1083.065,360.325,-95.646,176.508,27.016,154.537
C00938=1083.070,360.572,-95.682,176.511,27.022,154.538
C00939=1083.076,360.819,-95.718,176.515,27.028,154.539
C00940=1083.082,361.067,-95.754,176.518,27.033,154.540
C00941=1083.089,361.314,-95.790,176.522,27.039,154.541
C00942=1083.095,361.562,-95.826,176.525,27.044,154.542
C00943=1083.101,361.809,-95.863,176.528,27.050,154.543
C00944=1083.107,362.057,-95.898,176.531,27.056,154.544
C00945=1083.113,362.304,-95.935,176.534,27.062,154.545
C00946=1083.119,362.551,-95.970,176.538,27.067,154.546
C00947=1083.125,362.798,-96.007,176.541,27.073,154.547
C00948=1083.131,363.045,-96.043,176.544,27.079,154.548
C00949=1083.137,363.292,-96.079,176.547,27.084,154.549
C00950=1083.144,363.539,-96.115,176.551,27.090,154.550
C00951=1083.150,363.787,-96.151,176.554,27.096,154.551
C00952=1083.155,364.034,-96.188,176.558,27.102,154.552
C00953=1083.162,364.281,-96.224,176.560,27.108,154.554
C00954=1083.168,364.529,-96.261,176.564,27.114,154.555
C00955=1083.174,364.776,-96.297,176.567,27.120,154.556
C00956=1083.181,365.023,-96.333,176.571,27.126,154.557
C00957=1083.187,365.270,-96.369,176.574,27.131,154.558
C00958=1083.192,365.518,-96.406,176.577,27.137,154.559
C00959=1083.198,365.765,-96.442,176.580,27.143,154.560
C00960=1083.205,366.012,-96.479,176.584,27.149,154.561
C00961=1083.211,366.259,-96.515,176.587,27.155,154.562
C00962=1083.217,366.507,-96.552,176.591,27.161,154.563
C00963=1083.223,366.754,-96.589,176.594,27.167,154.564
C00964=1083.229,367.001,-96.625,176.597,27.173,154.565
C00965=1083.235,367.248,-96.662,176.601,27.179,154.566
C00966=1083.241,367.495,-96.698,176.604,27.185,154.567
C00967=1083.248,367.742,-96.735,176.608,27.191,154.568
C00968=1083.253,367.990,-96.772,176.610,27.197,154.569
C00969=1083.260,368.237,-96.808,176.614,27.203,154.570
C00970=1083.265,368.484,-96.845,176.617,27.209,154.572
C00971=1083.272,368.731,-96.882,176.621,27.215,154.573
C00972=1083.278,368.978,-96.918,176.623,27.221,154.574
C00973=1083.283,369.226,-96.955,176.627,27.227,154.575
C00974=1083.290,369.473,-96.992,176.631,27.233,154.576
C00975=1083.295,369.720,-97.029,176.634,27.239,154.577
C00976=1083.302,369.967,-97.065,176.637,27.245,154.578
C00977=1083.309,370.214,-97.103,176.640,27.251,154.579
C00978=1083.314,370.426,-97.134,176.643,27.257,154.580
C00979=1083.319,370.638,-97.166,176.646,27.262,154.581
C00980=1083.324,370.850,-97.198,176.649,27.267,154.582
C00981=1083.329,371.062,-97.230,176.652,27.272,154.583
C00982=1083.335,371.273,-97.260,176.655,27.278,154.584
C00983=1083.340,371.485,-97.293,176.658,27.283,154.585
C00984=1083.346,371.698,-97.324,176.661,27.288,154.586
C00985=1083.350,371.909,-97.356,176.664,27.293,154.587
C00986=1083.357,372.156,-97.393,176.667,27.300,154.588
C00987=1083.363,372.404,-97.430,176.670,27.306,154.589
C00988=1083.370,372.651,-97.467,176.674,27.313,154.590
C00989=1083.376,372.898,-97.504,176.677,27.318,154.591
C00990=1083.382,373.145,-97.541,176.680,27.325,154.592
C00991=1083.388,373.391,-97.579,176.684,27.331,154.594
C00992=1083.395,373.639,-97.615,176.687,27.337,154.595
C00993=1083.400,373.887,-97.653,176.691,27.344,154.596
C00994=1083.407,374.133,-97.690,176.693,27.350,154.597
C00995=1083.413,374.380,-97.727,176.697,27.356,154.598
C00996=1083.419,374.628,-97.765,176.701,27.363,154.599
C00997=1083.425,374.875,-97.803,176.704,27.369,154.601
C00998=1083.431,375.122,-97.839,176.707,27.375,154.602
C00999=1083.437,375.368,-97.877,176.711,27.382,154.603
C01000=1083.443,375.616,-97.914,176.714,27.388,154.604
C01001=1083.450,375.863,-97.951,176.718,27.395,154.605
C01002=1083.456,376.110,-97.989,176.721,27.401,154.606
C01003=1083.462,376.357,-98.026,176.724,27.408,154.608
C01004=1083.467,376.604,-98.064,176.728,27.415,154.609
C01005=1083.475,376.851,-98.101,176.731,27.421,154.610
C01006=1083.481,377.098,-98.139,176.734,27.427,154.611
C01007=1083.486,377.345,-98.176,176.738,27.434,154.613
C01008=1083.493,377.592,-98.214,176.742,27.441,154.614
C01009=1083.499,377.839,-98.252,176.744,27.447,154.615
C01010=1083.505,378.086,-98.289,176.748,27.454,154.616
C01011=1083.512,378.333,-98.327,176.752,27.460,154.617
C01012=1083.518,378.580,-98.365,176.754,27.467,154.619
C01013=1083.523,378.827,-98.402,176.758,27.473,154.620
C01014=1083.530,379.074,-98.440,176.762,27.480,154.621
C01015=1083.536,379.321,-98.477,176.765,27.487,154.622
C01016=1083.542,379.568,-98.515,176.768,27.493,154.624
C01017=1083.549,379.815,-98.553,176.772,27.500,154.625
C01018=1083.555,380.062,-98.591,176.776,27.506,154.626
C01019=1083.561,380.309,-98.629,176.779,27.513,154.627
C01020=1083.568,380.556,-98.666,176.782,27.520,154.629
C01021=1083.574,380.803,-98.705,176.786,27.527,154.630
C01022=1083.580,381.050,-98.742,176.789,27.533,154.631
C01023=1083.586,381.297,-98.780,176.793,27.540,154.632
C01024=1083.593,381.544,-98.819,176.796,27.547,154.634
C01025=1083.599,381.790,-98.857,176.800,27.554,154.635
C01026=1083.605,382.038,-98.895,176.803,27.561,154.636
C01027=1083.611,382.284,-98.932,176.807,27.568,154.637
C01028=1083.618,382.532,-98.971,176.810,27.574,154.639
C01029=1083.624,382.779,-99.008,176.813,27.581,154.640
C01030=1083.631,383.025,-99.047,176.817,27.588,154.641
C01031=1083.636,383.272,-99.085,176.821,27.595,154.643
C01032=1083.643,383.520,-99.123,176.823,27.602,154.644
C01033=1083.649,383.766,-99.162,176.827,27.609,154.645
C01034=1083.655,383.992,-99.197,176.831,27.615,154.647
C01035=1083.660,384.218,-99.232,176.833,27.622,154.648
C01036=1083.666,384.444,-99.267,176.836,27.628,154.649
C01037=1083.672,384.669,-99.302,176.840,27.635,154.650
C01038=1083.677,384.895,-99.337,176.843,27.641,154.651
C01039=1083.683,385.122,-99.372,176.847,27.647,154.653
C01040=1083.689,385.348,-99.407,176.849,27.654,154.654
C01041=1083.695,385.574,-99.442,176.852,27.660,154.655
C01042=1083.700,385.822,-99.481,176.856,27.668,154.657
C01043=1083.707,386.068,-99.519,176.859,27.675,154.658
C01044=1083.713,386.315,-99.558,176.863,27.682,154.659
C01045=1083.719,386.561,-99.596,176.867,27.689,154.661
C01046=1083.726,386.808,-99.635,176.870,27.696,154.662
C01047=1083.733,387.056,-99.673,176.874,27.703,154.663
C01048=1083.738,387.302,-99.712,176.877,27.711,154.665
C01049=1083.745,387.549,-99.751,176.880,27.718,154.666
C01050=1083.751,387.796,-99.788,176.884,27.725,154.668
C01051=1083.758,388.042,-99.827,176.888,27.732,154.669
C01052=1083.764,388.290,-99.867,176.891,27.740,154.670
C01053=1083.770,388.536,-99.904,176.895,27.747,154.672
C01054=1083.776,388.783,-99.943,176.898,27.754,154.673
C01055=1083.783,389.030,-99.982,176.902,27.762,154.675
C01056=1083.789,389.276,-100.021,176.905,27.769,154.676
C01057=1083.796,389.523,-100.060,176.908,27.776,154.677
C01058=1083.802,389.771,-100.098,176.912,27.783,154.679
C01059=1083.809,390.017,-100.137,176.916,27.791,154.680
C01060=1083.814,390.264,-100.176,176.919,27.798,154.682
C01061=1083.821,390.511,-100.215,176.923,27.805,154.683
C01062=1083.828,390.758,-100.254,176.927,27.813,154.685
C01063=1083.834,391.005,-100.293,176.930,27.820,154.686
C01064=1083.840,391.251,-100.332,176.934,27.828,154.687
C01065=1083.847,391.498,-100.370,176.937,27.835,154.689
C01066=1083.853,391.745,-100.410,176.941,27.843,154.690
C01067=1083.860,391.992,-100.449,176.945,27.850,154.692
C01068=1083.865,392.238,-100.488,176.948,27.858,154.693
C01069=1083.872,392.485,-100.527,176.952,27.866,154.695
C01070=1083.878,392.732,-100.566,176.956,27.873,154.696
C01071=1083.885,392.979,-100.605,176.958,27.881,154.698
C01072=1083.892,393.225,-100.645,176.962,27.888,154.699
C01073=1083.898,393.472,-100.684,176.965,27.896,154.701
C01074=1083.904,393.719,-100.723,176.969,27.904,154.702
C01075=1083.911,393.965,-100.762,176.973,27.911,154.704
C01076=1083.917,394.213,-100.801,176.976,27.919,154.705
C01077=1083.924,394.459,-100.841,176.980,27.927,154.707
C01078=1083.930,394.706,-100.880,176.983,27.934,154.708
C01079=1083.936,394.953,-100.920,176.987,27.942,154.710
C01080=1083.943,395.199,-100.959,176.991,27.950,154.711
C01081=1083.949,395.446,-100.999,176.994,27.958,154.713
C01082=1083.955,395.693,-101.038,176.998,27.966,154.715
C01083=1083.962,395.939,-101.077,177.001,27.974,154.716
C01084=1083.968,396.186,-101.117,177.005,27.982,154.718
C01085=1083.974,396.433,-101.157,177.008,27.989,154.719
C01086=1083.981,396.679,-101.196,177.012,27.998,154.721
C01087=1083.987,396.926,-101.236,177.016,28.005,154.722
C01088=1083.993,397.173,-101.275,177.019,28.013,154.724
C01089=1084.000,397.420,-101.315,177.023,28.022,154.726
C01090=1084.006,397.653,-101.352,177.026,28.029,154.727
C01091=1084.013,397.886,-101.390,177.030,28.037,154.729
C01092=1084.018,398.119,-101.427,177.034,28.044,154.730
C01093=1084.025,398.352,-101.465,177.036,28.052,154.732
C01094=1084.030,398.585,-101.502,177.040,28.059,154.733
C01095=1084.037,398.818,-101.540,177.044,28.067,154.735
C01096=1084.043,399.051,-101.577,177.047,28.075,154.736
C01097=1084.049,399.284,-101.615,177.051,28.083,154.738
C01098=1084.055,399.530,-101.655,177.054,28.091,154.739
C01099=1084.061,399.777,-101.695,177.058,28.099,154.741
C01100=1084.067,400.024,-101.735,177.062,28.107,154.743
C01101=1084.074,400.270,-101.775,177.065,28.116,154.744
C01102=1084.082,400.517,-101.815,177.069,28.124,154.746
C01103=1084.088,400.764,-101.855,177.072,28.132,154.748
C01104=1084.094,401.011,-101.895,177.076,28.140,154.750
C01105=1084.100,401.257,-101.935,177.079,28.149,154.751
C01106=1084.107,401.504,-101.975,177.084,28.157,154.753
C01107=1084.113,401.750,-102.015,177.087,28.165,154.755
C01108=1084.120,401.997,-102.055,177.091,28.174,154.756
C01109=1084.127,402.244,-102.096,177.094,28.182,154.758
C01110=1084.133,402.491,-102.136,177.098,28.191,154.760
C01111=1084.139,402.737,-102.176,177.102,28.199,154.761
C01112=1084.146,402.984,-102.216,177.106,28.208,154.763
C01113=1084.152,403.230,-102.256,177.110,28.216,154.765
C01114=1084.159,403.477,-102.297,177.113,28.225,154.767
C01115=1084.165,403.724,-102.337,177.117,28.234,154.768
C01116=1084.172,403.971,-102.377,177.120,28.242,154.770
C01117=1084.178,404.217,-102.419,177.125,28.251,154.772
C01118=1084.185,404.464,-102.459,177.128,28.260,154.774
C01119=1084.191,404.710,-102.499,177.132,28.268,154.775
C01120=1084.197,404.957,-102.539,177.135,28.277,154.777
C01121=1084.205,405.204,-102.581,177.139,28.285,154.779
C01122=1084.211,405.450,-102.621,177.143,28.294,154.781
C01123=1084.217,405.697,-102.662,177.147,28.303,154.782
C01124=1084.224,405.944,-102.702,177.150,28.312,154.784
C01125=1084.230,406.190,-102.743,177.154,28.321,154.786
C01126=1084.237,406.437,-102.783,177.158,28.330,154.788
C01127=1084.243,406.683,-102.825,177.162,28.338,154.790
C01128=1084.250,406.930,-102.865,177.165,28.347,154.792
C01129=1084.256,407.176,-102.906,177.170,28.357,154.793
C01130=1084.263,407.423,-102.946,177.173,28.365,154.795
C01131=1084.269,407.669,-102.988,177.177,28.374,154.797
C01132=1084.276,407.916,-103.028,177.180,28.383,154.799
C01133=1084.282,408.163,-103.070,177.185,28.393,154.801
C01134=1084.289,408.409,-103.110,177.188,28.401,154.803
C01135=1084.296,408.656,-103.151,177.192,28.411,154.805
C01136=1084.302,408.903,-103.192,177.196,28.420,154.807
C01137=1084.308,409.149,-103.233,177.200,28.429,154.808
C01138=1084.315,409.395,-103.275,177.203,28.438,154.810
C01139=1084.322,409.641,-103.316,177.208,28.448,154.812
C01140=1084.328,409.889,-103.357,177.211,28.457,154.814
C01141=1084.334,410.135,-103.398,177.216,28.466,154.816
C01142=1084.341,410.382,-103.439,177.219,28.475,154.818
C01143=1084.348,410.628,-103.480,177.223,28.485,154.820
C01144=1084.354,410.874,-103.522,177.227,28.494,154.822
C01145=1084.361,411.121,-103.562,177.231,28.503,154.824
C01146=1084.367,411.355,-103.602,177.234,28.512,154.826
C01147=1084.373,411.588,-103.641,177.238,28.521,154.828
C01148=1084.379,411.823,-103.680,177.242,28.530,154.829
C01149=1084.386,412.056,-103.719,177.246,28.539,154.831
C01150=1084.392,412.290,-103.759,177.249,28.548,154.833
C01151=1084.399,412.524,-103.798,177.253,28.557,154.835
C01152=1084.404,412.758,-103.837,177.257,28.566,154.837
C01153=1084.411,412.991,-103.877,177.261,28.575,154.839
C01154=1084.418,413.238,-103.918,177.265,28.585,154.841
C01155=1084.425,413.484,-103.959,177.269,28.594,154.843
C01156=1084.431,413.731,-104.001,177.273,28.604,154.845
C01157=1084.439,413.978,-104.042,177.277,28.614,154.847
C01158=1084.445,414.224,-104.084,177.281,28.623,154.849
C01159=1084.451,414.470,-104.126,177.285,28.633,154.851
C01160=1084.459,414.717,-104.168,177.288,28.643,154.853
C01161=1084.465,414.963,-104.209,177.293,28.653,154.855
C01162=1084.472,415.209,-104.250,177.296,28.662,154.857
C01163=1084.479,415.456,-104.293,177.301,28.672,154.859
C01164=1084.485,415.703,-104.335,177.304,28.682,154.861
C01165=1084.492,415.949,-104.376,177.309,28.692,154.863
C01166=1084.499,416.195,-104.418,177.312,28.702,154.865
C01167=1084.505,416.442,-104.460,177.317,28.712,154.868
C01168=1084.512,416.688,-104.502,177.321,28.722,154.870
C01169=1084.518,416.934,-104.544,177.325,28.732,154.872
C01170=1084.525,417.181,-104.586,177.329,28.742,154.874
C01171=1084.532,417.427,-104.628,177.332,28.752,154.876
C01172=1084.539,417.673,-104.670,177.337,28.763,154.878
C01173=1084.545,417.919,-104.712,177.341,28.773,154.881
C01174=1084.552,418.166,-104.754,177.345,28.783,154.883
C01175=1084.559,418.412,-104.797,177.349,28.793,154.885
C01176=1084.566,418.658,-104.839,177.354,28.804,154.887
C01177=1084.572,418.905,-104.881,177.357,28.814,154.889
C01178=1084.579,419.151,-104.923,177.362,28.824,154.891
C01179=1084.585,419.397,-104.966,177.366,28.835,154.894
C01180=1084.592,419.644,-105.008,177.369,28.845,154.896
C01181=1084.599,419.890,-105.050,177.374,28.856,154.898
C01182=1084.606,420.137,-105.093,177.378,28.866,154.900
C01183=1084.613,420.383,-105.135,177.383,28.877,154.903
C01184=1084.620,420.629,-105.177,177.386,28.887,154.905
C01185=1084.627,420.875,-105.220,177.391,28.898,154.907
C01186=1084.634,421.122,-105.262,177.395,28.908,154.909
C01187=1084.641,421.368,-105.305,177.399,28.919,154.912
C01188=1084.648,421.614,-105.347,177.403,28.929,154.914
C01189=1084.654,421.860,-105.390,177.407,28.940,154.916
C01190=1084.661,422.107,-105.432,177.412,28.951,154.918
C01191=1084.668,422.353,-105.475,177.416,28.961,154.921
C01192=1084.674,422.599,-105.518,177.420,28.972,154.923
C01193=1084.681,422.845,-105.561,177.424,28.983,154.925
C01194=1084.688,423.091,-105.604,177.428,28.994,154.928
C01195=1084.694,423.337,-105.646,177.433,29.005,154.930
C01196=1084.701,423.583,-105.689,177.437,29.016,154.933
C01197=1084.708,423.829,-105.732,177.442,29.027,154.935
C01198=1084.715,424.076,-105.775,177.445,29.038,154.937
C01199=1084.721,424.322,-105.818,177.449,29.049,154.940
C01200=1084.729,424.568,-105.861,177.454,29.060,154.942
C01201=1084.735,424.815,-105.904,177.458,29.071,154.944
C01202=1084.742,425.056,-105.946,177.463,29.082,154.947
C01203=1084.749,425.298,-105.989,177.467,29.094,154.949
C01204=1084.755,425.539,-106.031,177.471,29.104,154.952
C01205=1084.762,425.781,-106.074,177.475,29.115,154.954
C01206=1084.770,426.023,-106.116,177.479,29.126,154.957
C01207=1084.775,426.265,-106.158,177.484,29.138,154.959
C01208=1084.783,426.506,-106.200,177.488,29.149,154.961
C01209=1084.790,426.748,-106.243,177.492,29.160,154.964
C01210=1084.797,426.994,-106.287,177.496,29.171,154.966
C01211=1084.803,427.241,-106.330,177.501,29.183,154.969
C01212=1084.811,427.487,-106.373,177.505,29.194,154.971
C01213=1084.818,427.733,-106.417,177.509,29.206,154.974
C01214=1084.824,427.979,-106.460,177.514,29.217,154.976
C01215=1084.831,428.225,-106.503,177.518,29.229,154.979
C01216=1084.839,428.471,-106.547,177.523,29.240,154.981
C01217=1084.845,428.717,-106.590,177.527,29.252,154.984
C01218=1084.852,428.963,-106.634,177.532,29.264,154.987
C01219=1084.859,429.209,-106.678,177.536,29.276,154.989
C01220=1084.867,429.455,-106.721,177.540,29.287,154.992
C01221=1084.873,429.701,-106.765,177.545,29.299,154.994
C01222=1084.880,429.947,-106.809,177.549,29.312,154.997
C01223=1084.887,430.193,-106.852,177.555,29.323,155.000
C01224=1084.894,430.440,-106.896,177.559,29.336,155.002
C01225=1084.901,430.685,-106.940,177.563,29.348,155.005
C01226=1084.908,430.931,-106.984,177.568,29.360,155.008
C01227=1084.915,431.177,-107.028,177.572,29.372,155.010
C01228=1084.922,431.423,-107.072,177.577,29.384,155.013
C01229=1084.929,431.670,-107.116,177.581,29.396,155.016
C01230=1084.936,431.915,-107.160,177.585,29.408,155.018
C01231=1084.943,432.161,-107.204,177.590,29.420,155.021
C01232=1084.950,432.407,-107.247,177.595,29.432,155.024
C01233=1084.958,432.653,-107.292,177.600,29.445,155.027
C01234=1084.964,432.899,-107.336,177.604,29.458,155.029
C01235=1084.971,433.144,-107.381,177.608,29.470,155.032
C01236=1084.978,433.391,-107.425,177.613,29.482,155.035
C01237=1084.985,433.636,-107.469,177.617,29.495,155.038
C01238=1084.992,433.883,-107.513,177.623,29.507,155.040
C01239=1084.999,434.128,-107.558,177.627,29.520,155.043
C01240=1085.007,434.374,-107.603,177.632,29.532,155.046
C01241=1085.013,434.620,-107.646,177.636,29.545,155.049
C01242=1085.020,434.866,-107.691,177.641,29.558,155.052
C01243=1085.028,435.111,-107.735,177.646,29.571,155.055
C01244=1085.035,435.357,-107.780,177.650,29.584,155.057
C01245=1085.042,435.603,-107.824,177.655,29.597,155.060
C01246=1085.049,435.849,-107.869,177.660,29.609,155.063
C01247=1085.056,436.095,-107.914,177.664,29.622,155.066
C01248=1085.063,436.341,-107.959,177.669,29.635,155.069
C01249=1085.070,436.587,-108.003,177.674,29.649,155.072
C01250=1085.077,436.832,-108.048,177.679,29.662,155.075
C01251=1085.084,437.078,-108.093,177.683,29.675,155.078
C01252=1085.091,437.323,-108.137,177.688,29.688,155.081
C01253=1085.098,437.570,-108.182,177.693,29.701,155.084
C01254=1085.106,437.815,-108.227,177.697,29.714,155.087
C01255=1085.113,438.061,-108.271,177.703,29.728,155.090
C01256=1085.120,438.307,-108.316,177.707,29.741,155.093
C01257=1085.128,438.552,-108.362,177.712,29.754,155.096
C01258=1085.140,438.956,-108.436,177.720,29.776,155.101
C01259=1085.151,439.360,-108.510,177.728,29.799,155.106
C01260=1085.164,439.763,-108.584,177.736,29.821,155.111
C01261=1085.176,440.167,-108.658,177.744,29.843,155.116
C01262=1085.183,440.413,-108.704,177.749,29.857,155.119
C01263=1085.190,440.659,-108.749,177.754,29.871,155.122
C01264=1085.197,440.904,-108.795,177.759,29.885,155.125
C01265=1085.204,441.150,-108.840,177.764,29.899,155.129
C01266=1085.212,441.396,-108.885,177.768,29.913,155.132
C01267=1085.219,441.641,-108.931,177.774,29.927,155.135
C01268=1085.226,441.887,-108.976,177.778,29.941,155.138
C01269=1085.234,442.133,-109.022,177.784,29.955,155.141
C01270=1085.242,442.378,-109.068,177.788,29.969,155.145
C01271=1085.249,442.624,-109.114,177.794,29.984,155.148
C01272=1085.256,442.870,-109.159,177.798,29.997,155.151
C01273=1085.263,443.115,-109.205,177.804,30.012,155.154
C01274=1085.270,443.360,-109.250,177.809,30.027,155.158
C01275=1085.277,443.606,-109.296,177.814,30.041,155.161
C01276=1085.284,443.852,-109.342,177.819,30.055,155.164
C01277=1085.292,444.097,-109.388,177.824,30.070,155.168
C01278=1085.300,444.342,-109.434,177.829,30.084,155.171
C01279=1085.307,444.588,-109.480,177.834,30.099,155.174
C01280=1085.315,444.834,-109.526,177.840,30.114,155.178
C01281=1085.322,445.080,-109.571,177.844,30.128,155.181
C01282=1085.330,445.325,-109.618,177.850,30.143,155.185
C01283=1085.337,445.570,-109.664,177.854,30.158,155.188
C01284=1085.344,445.816,-109.710,177.859,30.173,155.192
C01285=1085.351,446.061,-109.757,177.863,30.188,155.195
C01286=1085.359,446.307,-109.803,177.867,30.202,155.198
C01287=1085.366,446.552,-109.849,177.871,30.217,155.202
C01288=1085.374,446.797,-109.896,177.875,30.232,155.206
C01289=1085.381,447.044,-109.942,177.879,30.246,155.209
C01290=1085.389,447.289,-109.988,177.881,30.261,155.213
C01291=1085.396,447.534,-110.035,177.885,30.275,155.216
C01292=1085.403,447.780,-110.081,177.887,30.290,155.220
C01293=1085.412,448.025,-110.128,177.890,30.305,155.223
C01294=1085.419,448.271,-110.175,177.893,30.320,155.227
C01295=1085.426,448.516,-110.220,177.895,30.334,155.230
C01296=1085.434,448.761,-110.267,177.897,30.348,155.234
C01297=1085.441,449.008,-110.314,177.899,30.363,155.237
C01298=1085.449,449.252,-110.360,177.900,30.377,155.241
C01299=1085.456,449.496,-110.406,177.902,30.392,155.245
C01300=1085.466,449.742,-110.453,177.904,30.406,155.248
C01301=1085.477,449.988,-110.497,177.905,30.419,155.251
C01302=1085.103,449.981,-110.702,177.871,30.601,155.300
C01303=1085.092,449.735,-110.657,177.869,30.589,155.297
C01304=1085.082,449.489,-110.612,177.868,30.575,155.294
C01305=1085.074,449.244,-110.566,177.866,30.560,155.290
C01306=1085.067,448.999,-110.519,177.864,30.546,155.287
C01307=1085.059,448.754,-110.473,177.862,30.531,155.283
C01308=1085.051,448.508,-110.425,177.859,30.517,155.279
C01309=1085.044,448.263,-110.379,177.857,30.502,155.276
C01310=1085.036,448.018,-110.333,177.855,30.487,155.272
C01311=1085.029,447.773,-110.286,177.851,30.473,155.269
C01312=1085.022,447.526,-110.239,177.849,30.458,155.265
C01313=1085.014,447.282,-110.193,177.846,30.443,155.262
C01314=1085.007,447.036,-110.147,177.842,30.429,155.258
C01315=1084.998,446.790,-110.100,177.839,30.414,155.255
C01316=1084.991,446.545,-110.054,177.835,30.399,155.251
C01317=1084.984,446.299,-110.007,177.831,30.384,155.248
C01318=1084.977,446.054,-109.961,177.827,30.370,155.244
C01319=1084.969,445.809,-109.914,177.822,30.355,155.241
C01320=1084.962,445.563,-109.868,177.817,30.340,155.237
C01321=1084.955,445.318,-109.822,177.813,30.325,155.234
C01322=1084.946,445.072,-109.775,177.807,30.311,155.230
C01323=1084.939,444.826,-109.729,177.803,30.296,155.227
C01324=1084.932,444.581,-109.684,177.797,30.281,155.224
C01325=1084.925,444.335,-109.637,177.791,30.266,155.220
C01326=1084.917,444.090,-109.592,177.787,30.252,155.217
C01327=1084.910,443.844,-109.546,177.781,30.237,155.213
C01328=1084.903,443.599,-109.500,177.776,30.223,155.210
C01329=1084.895,443.353,-109.454,177.771,30.208,155.207
C01330=1084.887,443.108,-109.408,177.766,30.194,155.203
C01331=1084.880,442.862,-109.362,177.761,30.179,155.200
C01332=1084.873,442.617,-109.317,177.755,30.165,155.197
C01333=1084.865,442.371,-109.271,177.750,30.151,155.194
C01334=1084.858,442.125,-109.225,177.745,30.137,155.190
C01335=1084.851,441.880,-109.179,177.740,30.123,155.187
C01336=1084.843,441.635,-109.133,177.735,30.109,155.184
C01337=1084.836,441.388,-109.088,177.730,30.095,155.181
C01338=1084.829,441.143,-109.042,177.725,30.081,155.178
C01339=1084.821,440.897,-108.997,177.720,30.067,155.174
C01340=1084.814,440.652,-108.952,177.715,30.053,155.171
C01341=1084.807,440.407,-108.906,177.710,30.039,155.168
C01342=1084.800,440.160,-108.861,177.705,30.025,155.165
C01343=1084.789,439.771,-108.789,177.697,30.003,155.160
C01344=1084.776,439.382,-108.717,177.690,29.982,155.155
C01345=1084.765,438.993,-108.646,177.681,29.960,155.150
C01346=1084.753,438.604,-108.574,177.673,29.939,155.145
C01347=1084.746,438.358,-108.529,177.669,29.926,155.142
C01348=1084.739,438.113,-108.485,177.663,29.912,155.139
C01349=1084.731,437.867,-108.439,177.659,29.899,155.136
C01350=1084.724,437.621,-108.394,177.654,29.886,155.133
C01351=1084.717,437.375,-108.349,177.649,29.873,155.130
C01352=1084.710,437.130,-108.305,177.644,29.859,155.127
C01353=1084.703,436.884,-108.260,177.640,29.846,155.124
C01354=1084.695,436.638,-108.215,177.634,29.833,155.121
C01355=1084.689,436.392,-108.170,177.630,29.820,155.118
C01356=1084.681,436.146,-108.125,177.625,29.807,155.115
C01357=1084.674,435.900,-108.080,177.620,29.794,155.113
C01358=1084.666,435.655,-108.036,177.615,29.781,155.110
C01359=1084.659,435.409,-107.992,177.611,29.768,155.107
C01360=1084.652,435.164,-107.947,177.606,29.755,155.104
C01361=1084.645,434.918,-107.902,177.601,29.742,155.101
C01362=1084.639,434.672,-107.858,177.596,29.730,155.098
C01363=1084.631,434.426,-107.813,177.592,29.717,155.095
C01364=1084.624,434.179,-107.768,177.587,29.704,155.092
C01365=1084.617,433.934,-107.724,177.583,29.692,155.090
C01366=1084.610,433.688,-107.680,177.577,29.679,155.087
C01367=1084.603,433.442,-107.636,177.573,29.666,155.084
C01368=1084.596,433.196,-107.592,177.568,29.654,155.081
C01369=1084.589,432.950,-107.547,177.564,29.641,155.078
C01370=1084.582,432.705,-107.502,177.559,29.629,155.076
C01371=1084.574,432.459,-107.459,177.555,29.617,155.073
C01372=1084.568,432.213,-107.415,177.549,29.604,155.070
C01373=1084.561,431.967,-107.370,177.545,29.592,155.067
C01374=1084.554,431.721,-107.327,177.540,29.580,155.065
C01375=1084.546,431.474,-107.282,177.536,29.568,155.062
C01376=1084.540,431.229,-107.238,177.531,29.555,155.059
C01377=1084.532,430.983,-107.194,177.527,29.543,155.057
C01378=1084.526,430.737,-107.150,177.522,29.531,155.054
C01379=1084.518,430.492,-107.106,177.518,29.519,155.051
C01380=1084.511,430.245,-107.062,177.513,29.507,155.049
C01381=1084.505,429.999,-107.018,177.509,29.495,155.046
C01382=1084.497,429.753,-106.975,177.503,29.483,155.043
C01383=1084.490,429.507,-106.931,177.499,29.471,155.041
C01384=1084.483,429.261,-106.888,177.494,29.459,155.038
C01385=1084.477,429.015,-106.844,177.490,29.448,155.036
C01386=1084.469,428.769,-106.800,177.486,29.436,155.033
C01387=1084.463,428.523,-106.756,177.481,29.424,155.030
C01388=1084.456,428.277,-106.713,177.477,29.412,155.028
C01389=1084.449,428.031,-106.669,177.472,29.401,155.025
C01390=1084.441,427.785,-106.625,177.468,29.389,155.023
C01391=1084.434,427.539,-106.582,177.463,29.377,155.020
C01392=1084.428,427.293,-106.538,177.459,29.366,155.018
C01393=1084.420,427.046,-106.495,177.455,29.355,155.015
C01394=1084.413,426.800,-106.452,177.451,29.343,155.013
C01395=1084.406,426.558,-106.409,177.446,29.332,155.010
C01396=1084.400,426.316,-106.367,177.442,29.321,155.008
C01397=1084.393,426.073,-106.324,177.437,29.310,155.005
C01398=1084.386,425.831,-106.281,177.433,29.298,155.003
C01399=1084.379,425.589,-106.239,177.428,29.287,155.001
C01400=1084.372,425.346,-106.197,177.424,29.276,154.998
C01401=1084.366,425.104,-106.154,177.420,29.265,154.996
C01402=1084.359,424.862,-106.111,177.415,29.254,154.993
C01403=1084.352,424.615,-106.068,177.411,29.243,154.991
C01404=1084.345,424.369,-106.025,177.407,29.232,154.988
C01405=1084.338,424.123,-105.983,177.403,29.221,154.986
C01406=1084.331,423.877,-105.939,177.398,29.210,154.984
C01407=1084.324,423.631,-105.896,177.394,29.199,154.981
C01408=1084.318,423.384,-105.854,177.390,29.188,154.979
C01409=1084.310,423.139,-105.811,177.385,29.177,154.977
C01410=1084.304,422.892,-105.767,177.381,29.166,154.974
C01411=1084.298,422.646,-105.725,177.377,29.155,154.972
C01412=1084.291,422.399,-105.682,177.373,29.144,154.970
C01413=1084.284,422.153,-105.640,177.368,29.133,154.967
C01414=1084.277,421.908,-105.597,177.364,29.122,154.965
C01415=1084.270,421.661,-105.554,177.360,29.112,154.962
C01416=1084.263,421.415,-105.511,177.356,29.101,154.960
C01417=1084.256,421.169,-105.469,177.351,29.090,154.958
C01418=1084.249,420.922,-105.426,177.347,29.080,154.956
C01419=1084.242,420.676,-105.384,177.343,29.070,154.953
C01420=1084.235,420.430,-105.341,177.339,29.059,154.951
C01421=1084.229,420.184,-105.299,177.334,29.048,154.949
C01422=1084.222,419.937,-105.256,177.330,29.038,154.947
C01423=1084.215,419.691,-105.214,177.326,29.027,154.944
C01424=1084.209,419.445,-105.171,177.322,29.017,154.942
C01425=1084.202,419.198,-105.130,177.317,29.006,154.940
C01426=1084.195,418.952,-105.087,177.314,28.996,154.938
C01427=1084.188,418.706,-105.045,177.309,28.986,154.936
C01428=1084.182,418.460,-105.002,177.305,28.976,154.933
C01429=1084.175,418.213,-104.960,177.301,28.965,154.931
C01430=1084.167,417.967,-104.918,177.297,28.955,154.929
C01431=1084.161,417.721,-104.876,177.293,28.945,154.927
C01432=1084.155,417.474,-104.834,177.289,28.934,154.925
C01433=1084.148,417.228,-104.792,177.284,28.924,154.922
C01434=1084.141,416.982,-104.749,177.281,28.914,154.920
C01435=1084.134,416.735,-104.707,177.276,28.904,154.918
C01436=1084.128,416.489,-104.665,177.272,28.894,154.916
C01437=1084.122,416.242,-104.623,177.268,28.884,154.914
C01438=1084.114,415.996,-104.581,177.263,28.874,154.912
C01439=1084.107,415.749,-104.540,177.260,28.864,154.910
C01440=1084.101,415.504,-104.497,177.255,28.854,154.908
C01441=1084.094,415.257,-104.456,177.252,28.845,154.906
C01442=1084.087,415.010,-104.414,177.247,28.834,154.903
C01443=1084.080,414.764,-104.372,177.244,28.825,154.901
C01444=1084.074,414.518,-104.331,177.239,28.815,154.899
C01445=1084.067,414.271,-104.289,177.236,28.805,154.897
C01446=1084.060,414.025,-104.248,177.231,28.795,154.895
C01447=1084.053,413.778,-104.205,177.228,28.786,154.893
C01448=1084.047,413.532,-104.164,177.223,28.776,154.891
C01449=1084.040,413.286,-104.123,177.220,28.766,154.889
C01450=1084.033,413.039,-104.081,177.215,28.757,154.887
C01451=1084.027,412.804,-104.041,177.212,28.748,154.885
C01452=1084.020,412.570,-104.003,177.208,28.739,154.883
C01453=1084.014,412.336,-103.963,177.204,28.730,154.881
C01454=1084.008,412.101,-103.924,177.200,28.720,154.879
C01455=1084.002,411.867,-103.883,177.196,28.712,154.878
C01456=1083.995,411.633,-103.844,177.192,28.702,154.876
C01457=1083.989,411.398,-103.806,177.189,28.693,154.874
C01458=1083.983,411.164,-103.766,177.185,28.685,154.872
C01459=1083.976,410.917,-103.725,177.181,28.675,154.870
C01460=1083.970,410.671,-103.684,177.177,28.666,154.868
C01461=1083.963,410.424,-103.642,177.174,28.656,154.866
C01462=1083.957,410.178,-103.601,177.169,28.647,154.864
C01463=1083.949,409.931,-103.560,177.166,28.638,154.862
C01464=1083.943,409.685,-103.518,177.162,28.629,154.860
C01465=1083.936,409.438,-103.478,177.157,28.619,154.858
C01466=1083.930,409.192,-103.436,177.154,28.610,154.857
C01467=1083.923,408.945,-103.395,177.150,28.601,154.855
C01468=1083.917,408.698,-103.354,177.146,28.592,154.853
C01469=1083.910,408.452,-103.313,177.142,28.582,154.851
C01470=1083.903,408.206,-103.272,177.139,28.573,154.849
C01471=1083.897,407.958,-103.231,177.134,28.564,154.847
C01472=1083.891,407.713,-103.190,177.131,28.555,154.845
C01473=1083.885,407.466,-103.149,177.127,28.546,154.843
C01474=1083.878,407.219,-103.108,177.123,28.537,154.841
C01475=1083.871,406.973,-103.067,177.119,28.528,154.840
C01476=1083.865,406.726,-103.027,177.115,28.519,154.838
C01477=1083.858,406.480,-102.985,177.112,28.511,154.836
C01478=1083.852,406.233,-102.945,177.107,28.501,154.834
C01479=1083.845,405.986,-102.905,177.104,28.492,154.832
C01480=1083.839,405.740,-102.863,177.100,28.484,154.830
C01481=1083.832,405.493,-102.823,177.097,28.475,154.829
C01482=1083.825,405.247,-102.782,177.092,28.466,154.827
C01483=1083.819,405.000,-102.742,177.088,28.457,154.825
C01484=1083.812,404.754,-102.702,177.085,28.449,154.823
C01485=1083.807,404.507,-102.661,177.081,28.440,154.821
C01486=1083.799,404.260,-102.620,177.078,28.431,154.820
C01487=1083.793,404.014,-102.579,177.073,28.422,154.818
C01488=1083.787,403.767,-102.539,177.070,28.414,154.816
C01489=1083.780,403.520,-102.499,177.066,28.405,154.814
C01490=1083.773,403.274,-102.459,177.062,28.397,154.813
C01491=1083.767,403.027,-102.419,177.059,28.388,154.811
C01492=1083.760,402.780,-102.378,177.054,28.379,154.809
C01493=1083.753,402.534,-102.337,177.051,28.371,154.807
C01494=1083.747,402.287,-102.297,177.047,28.362,154.806
C01495=1083.740,402.041,-102.257,177.043,28.354,154.804
C01496=1083.734,401.794,-102.217,177.040,28.346,154.802
C01497=1083.728,401.548,-102.177,177.036,28.337,154.801
C01498=1083.721,401.301,-102.136,177.033,28.329,154.799
C01499=1083.715,401.053,-102.097,177.029,28.321,154.797
C01500=1083.708,400.807,-102.056,177.024,28.312,154.796
C01501=1083.702,400.560,-102.016,177.021,28.304,154.794
C01502=1083.695,400.314,-101.976,177.017,28.295,154.792
C01503=1083.689,400.067,-101.936,177.014,28.287,154.790
C01504=1083.683,399.821,-101.896,177.010,28.279,154.789
C01505=1083.676,399.574,-101.855,177.006,28.271,154.787
C01506=1083.670,399.327,-101.816,177.003,28.262,154.785
C01507=1083.663,399.094,-101.778,176.999,28.255,154.784
C01508=1083.657,398.860,-101.741,176.996,28.247,154.782
C01509=1083.651,398.626,-101.703,176.993,28.239,154.781
C01510=1083.644,398.393,-101.665,176.989,28.232,154.779
C01511=1083.639,398.160,-101.627,176.985,28.224,154.778
C01512=1083.633,397.926,-101.590,176.982,28.216,154.776
C01513=1083.626,397.692,-101.552,176.978,28.209,154.775
C01514=1083.621,397.459,-101.514,176.975,28.201,154.773
C01515=1083.615,397.212,-101.475,176.972,28.193,154.772
C01516=1083.608,396.966,-101.435,176.968,28.185,154.770
C01517=1083.602,396.719,-101.396,176.964,28.177,154.768
C01518=1083.595,396.472,-101.356,176.961,28.169,154.767
C01519=1083.588,396.225,-101.317,176.957,28.161,154.765
C01520=1083.582,395.979,-101.277,176.954,28.154,154.764
C01521=1083.576,395.732,-101.237,176.950,28.146,154.762
C01522=1083.570,395.485,-101.197,176.946,28.137,154.760
C01523=1083.563,395.238,-101.158,176.943,28.130,154.759
C01524=1083.557,394.991,-101.119,176.939,28.122,154.757
C01525=1083.550,394.745,-101.079,176.935,28.114,154.756
C01526=1083.543,394.498,-101.040,176.932,28.106,154.754
C01527=1083.537,394.251,-101.000,176.928,28.098,154.753
C01528=1083.530,394.004,-100.961,176.924,28.091,154.751
C01529=1083.524,393.757,-100.921,176.921,28.083,154.750
C01530=1083.518,393.511,-100.883,176.917,28.075,154.748
C01531=1083.512,393.264,-100.844,176.913,28.068,154.747
C01532=1083.506,393.017,-100.804,176.910,28.060,154.745
C01533=1083.499,392.771,-100.765,176.906,28.052,154.744
C01534=1083.493,392.524,-100.725,176.903,28.045,154.742
C01535=1083.486,392.277,-100.686,176.899,28.037,154.741
C01536=1083.480,392.030,-100.647,176.895,28.029,154.739
C01537=1083.474,391.784,-100.608,176.892,28.022,154.738
C01538=1083.467,391.537,-100.570,176.888,28.014,154.736
C01539=1083.461,391.290,-100.530,176.884,28.007,154.735
C01540=1083.454,391.043,-100.491,176.882,28.000,154.733
C01541=1083.448,390.797,-100.453,176.878,27.992,154.732
C01542=1083.442,390.549,-100.413,176.874,27.985,154.730
C01543=1083.435,390.303,-100.375,176.871,27.977,154.729
C01544=1083.428,390.056,-100.336,176.867,27.970,154.728
C01545=1083.422,389.809,-100.297,176.863,27.962,154.726
C01546=1083.416,389.563,-100.258,176.860,27.955,154.725
C01547=1083.409,389.316,-100.219,176.856,27.947,154.723
C01548=1083.402,389.069,-100.180,176.852,27.940,154.722
C01549=1083.397,388.822,-100.142,176.849,27.933,154.720
C01550=1083.390,388.575,-100.103,176.846,27.926,154.719
C01551=1083.383,388.328,-100.064,176.842,27.918,154.718
C01552=1083.377,388.082,-100.026,176.838,27.911,154.716
C01553=1083.371,387.834,-99.987,176.835,27.904,154.715
C01554=1083.364,387.588,-99.948,176.831,27.897,154.713
C01555=1083.358,387.341,-99.910,176.827,27.889,154.712
C01556=1083.351,387.095,-99.871,176.824,27.882,154.711
C01557=1083.346,386.847,-99.832,176.821,27.875,154.709
C01558=1083.339,386.601,-99.794,176.817,27.868,154.708
C01559=1083.333,386.353,-99.755,176.814,27.861,154.706
C01560=1083.327,386.107,-99.717,176.810,27.853,154.705
C01561=1083.320,385.860,-99.678,176.806,27.846,154.704
C01562=1083.314,385.614,-99.640,176.803,27.839,154.702
C01563=1083.309,385.387,-99.604,176.800,27.832,154.701
C01564=1083.302,385.160,-99.569,176.797,27.826,154.700
C01565=1083.296,384.933,-99.534,176.793,27.820,154.699
C01566=1083.292,384.706,-99.499,176.790,27.813,154.697
C01567=1083.285,384.480,-99.464,176.787,27.807,154.696
C01568=1083.280,384.254,-99.429,176.784,27.800,154.695
C01569=1083.274,384.027,-99.393,176.781,27.794,154.694
C01570=1083.268,383.801,-99.359,176.777,27.787,154.692
C01571=1083.262,383.554,-99.319,176.773,27.780,154.691
C01572=1083.256,383.307,-99.282,176.771,27.773,154.690
C01573=1083.250,383.059,-99.244,176.767,27.766,154.688
C01574=1083.243,382.813,-99.205,176.763,27.759,154.687
C01575=1083.237,382.566,-99.167,176.760,27.752,154.686
C01576=1083.231,382.319,-99.129,176.757,27.746,154.684
C01577=1083.225,382.072,-99.091,176.753,27.739,154.683
C01578=1083.218,381.826,-99.053,176.749,27.732,154.682
C01579=1083.212,381.578,-99.014,176.746,27.725,154.681
C01580=1083.206,381.331,-98.977,176.743,27.718,154.679
C01581=1083.199,381.084,-98.939,176.739,27.712,154.678
C01582=1083.193,380.837,-98.901,176.735,27.705,154.677
C01583=1083.186,380.590,-98.863,176.732,27.698,154.675
C01584=1083.180,380.343,-98.826,176.729,27.691,154.674
C01585=1083.174,380.097,-98.788,176.725,27.685,154.673
C01586=1083.168,379.850,-98.749,176.722,27.678,154.672
C01587=1083.162,379.603,-98.711,176.719,27.671,154.670
C01588=1083.156,379.355,-98.674,176.715,27.665,154.669
C01589=1083.149,379.108,-98.637,176.711,27.658,154.668
C01590=1083.143,378.862,-98.599,176.708,27.651,154.667
C01591=1083.137,378.614,-98.561,176.705,27.645,154.666
C01592=1083.131,378.368,-98.523,176.701,27.638,154.664
C01593=1083.124,378.120,-98.485,176.697,27.631,154.663
C01594=1083.117,377.874,-98.448,176.695,27.625,154.662
C01595=1083.112,377.627,-98.410,176.691,27.618,154.661
C01596=1083.105,377.379,-98.372,176.687,27.611,154.659
C01597=1083.099,377.132,-98.335,176.684,27.605,154.658
C01598=1083.094,376.885,-98.297,176.681,27.598,154.657
C01599=1083.087,376.639,-98.260,176.677,27.592,154.656
C01600=1083.080,376.391,-98.222,176.674,27.585,154.654
C01601=1083.075,376.144,-98.185,176.670,27.579,154.653
C01602=1083.069,375.897,-98.147,176.667,27.572,154.652
C01603=1083.062,375.650,-98.109,176.664,27.566,154.651
C01604=1083.056,375.404,-98.072,176.660,27.559,154.650
C01605=1083.050,375.156,-98.035,176.656,27.553,154.649
C01606=1083.044,374.910,-97.998,176.654,27.546,154.647
C01607=1083.038,374.662,-97.960,176.650,27.540,154.646
C01608=1083.031,374.415,-97.922,176.647,27.534,154.645
C01609=1083.026,374.168,-97.885,176.643,27.527,154.644
C01610=1083.019,373.921,-97.848,176.639,27.521,154.643
C01611=1083.013,373.674,-97.810,176.637,27.515,154.641
C01612=1083.006,373.427,-97.774,176.633,27.508,154.640
C01613=1083.001,373.179,-97.737,176.629,27.502,154.639
C01614=1082.994,372.933,-97.699,176.626,27.496,154.638
C01615=1082.988,372.685,-97.662,176.623,27.489,154.637
C01616=1082.981,372.438,-97.625,176.620,27.483,154.636
C01617=1082.976,372.191,-97.588,176.616,27.477,154.635
C01618=1082.969,371.945,-97.551,176.612,27.471,154.633
C01619=1082.964,371.732,-97.519,176.609,27.465,154.632
C01620=1082.958,371.520,-97.487,176.607,27.460,154.631
C01621=1082.953,371.307,-97.456,176.604,27.455,154.630
C01622=1082.948,371.095,-97.424,176.601,27.449,154.629
C01623=1082.942,370.882,-97.392,176.598,27.444,154.629
C01624=1082.937,370.670,-97.361,176.595,27.439,154.628
C01625=1082.933,370.457,-97.328,176.592,27.434,154.627
C01626=1082.927,370.245,-97.297,176.589,27.428,154.626
C01627=1082.921,369.998,-97.260,176.586,27.422,154.625
C01628=1082.914,369.751,-97.223,176.583,27.416,154.623
C01629=1082.908,369.503,-97.186,176.579,27.410,154.622
C01630=1082.902,369.256,-97.149,176.576,27.404,154.621
C01631=1082.896,369.009,-97.112,176.572,27.398,154.620
C01632=1082.890,368.762,-97.076,176.570,27.392,154.619
C01633=1082.883,368.515,-97.039,176.566,27.386,154.618
C01634=1082.878,368.267,-97.002,176.563,27.380,154.617
C01635=1082.872,368.020,-96.966,176.559,27.374,154.616
C01636=1082.865,367.773,-96.929,176.555,27.367,154.615
C01637=1082.860,367.526,-96.892,176.553,27.361,154.614
C01638=1082.853,367.279,-96.856,176.549,27.355,154.613
C01639=1082.847,367.032,-96.819,176.546,27.349,154.611
C01640=1082.841,366.784,-96.782,176.542,27.343,154.610
C01641=1082.835,366.537,-96.746,176.539,27.338,154.609
C01642=1082.829,366.290,-96.709,176.536,27.331,154.608
C01643=1082.823,366.043,-96.672,176.533,27.325,154.607
C01644=1082.817,365.796,-96.636,176.529,27.319,154.606
C01645=1082.810,365.549,-96.599,176.526,27.314,154.605
C01646=1082.805,365.301,-96.562,176.522,27.307,154.604
C01647=1082.799,365.054,-96.527,176.519,27.302,154.603
C01648=1082.792,364.807,-96.490,176.516,27.296,154.602
C01649=1082.786,364.560,-96.454,176.513,27.290,154.601
C01650=1082.780,364.313,-96.417,176.509,27.284,154.600
C01651=1082.774,364.065,-96.382,176.506,27.279,154.599
C01652=1082.768,363.818,-96.345,176.502,27.273,154.598
C01653=1082.762,363.570,-96.308,176.499,27.267,154.597
C01654=1082.756,363.323,-96.272,176.496,27.261,154.596
C01655=1082.749,363.076,-96.236,176.493,27.255,154.595
C01656=1082.743,362.829,-96.199,176.489,27.249,154.594
C01657=1082.737,362.581,-96.164,176.486,27.244,154.593
C01658=1082.731,362.334,-96.127,176.483,27.238,154.592
C01659=1082.724,362.087,-96.091,176.479,27.232,154.591
C01660=1082.719,361.840,-96.056,176.477,27.227,154.590
C01661=1082.713,361.593,-96.019,176.473,27.221,154.589
C01662=1082.707,361.345,-95.983,176.470,27.215,154.588
C01663=1082.700,361.098,-95.947,176.466,27.209,154.587
C01664=1082.694,360.850,-95.911,176.463,27.204,154.586
C01665=1082.688,360.603,-95.875,176.459,27.198,154.585
C01666=1082.682,360.356,-95.839,176.456,27.192,154.584
C01667=1082.676,360.108,-95.803,176.454,27.187,154.583
C01668=1082.670,359.862,-95.767,176.450,27.181,154.582
C01669=1082.664,359.614,-95.731,176.447,27.175,154.581
C01670=1082.658,359.367,-95.695,176.443,27.169,154.580
C01671=1082.652,359.119,-95.659,176.440,27.164,154.579
C01672=1082.646,358.872,-95.624,176.436,27.159,154.578
C01673=1082.640,358.624,-95.588,176.433,27.153,154.577
C01674=1082.634,358.378,-95.552,176.430,27.148,154.576
C01675=1082.623,357.969,-95.493,176.424,27.138,154.574
C01676=1082.613,357.559,-95.434,176.419,27.129,154.573
C01677=1082.603,357.150,-95.375,176.414,27.120,154.571
C01678=1082.593,356.742,-95.316,176.409,27.111,154.570
C01679=1082.587,356.494,-95.280,176.405,27.105,154.569
C01680=1082.581,356.247,-95.245,176.402,27.100,154.568
C01681=1082.575,355.999,-95.209,176.398,27.095,154.567
C01682=1082.569,355.752,-95.174,176.395,27.089,154.566
C01683=1082.563,355.505,-95.138,176.393,27.084,154.565
C01684=1082.557,355.257,-95.102,176.389,27.078,154.564
C01685=1082.551,355.010,-95.067,176.386,27.073,154.563
C01686=1082.545,354.763,-95.032,176.383,27.068,154.562
C01687=1082.539,354.515,-94.996,176.379,27.062,154.561
C01688=1082.533,354.268,-94.961,176.376,27.057,154.560
C01689=1082.527,354.021,-94.925,176.373,27.051,154.559
C01690=1082.521,353.773,-94.890,176.369,27.046,154.558
C01691=1082.515,353.525,-94.854,176.367,27.040,154.557
C01692=1082.509,353.278,-94.819,176.363,27.035,154.557
C01693=1082.502,353.031,-94.784,176.360,27.030,154.556
C01694=1082.497,352.784,-94.748,176.357,27.024,154.555
C01695=1082.491,352.536,-94.712,176.353,27.019,154.554
C01696=1082.485,352.288,-94.678,176.350,27.013,154.553
C01697=1082.479,352.041,-94.642,176.347,27.009,154.552
C01698=1082.472,351.794,-94.608,176.343,27.003,154.551
C01699=1082.466,351.546,-94.572,176.340,26.998,154.550
C01700=1082.460,351.299,-94.538,176.337,26.993,154.549
C01701=1082.454,351.051,-94.502,176.335,26.987,154.548
C01702=1082.448,350.804,-94.466,176.331,26.982,154.548
C01703=1082.442,350.557,-94.431,176.328,26.977,154.547
C01704=1082.437,350.309,-94.396,176.325,26.972,154.546
C01705=1082.430,350.061,-94.361,176.321,26.966,154.545
C01706=1082.425,349.814,-94.327,176.318,26.961,154.544
C01707=1082.418,349.566,-94.292,176.315,26.956,154.543
C01708=1082.412,349.319,-94.256,176.311,26.951,154.542
C01709=1082.406,349.071,-94.222,176.308,26.945,154.541
C01710=1082.401,348.824,-94.186,176.305,26.941,154.541
C01711=1082.394,348.576,-94.152,176.302,26.935,154.540
C01712=1082.388,348.329,-94.116,176.299,26.930,154.539
C01713=1082.382,348.081,-94.082,176.296,26.925,154.538
C01714=1082.376,347.834,-94.046,176.293,26.920,154.537
C01715=1082.370,347.586,-94.012,176.289,26.915,154.536
C01716=1082.364,347.339,-93.977,176.286,26.910,154.535
C01717=1082.358,347.091,-93.943,176.283,26.904,154.535
C01718=1082.352,346.844,-93.908,176.280,26.899,154.534
C01719=1082.347,346.597,-93.873,176.276,26.894,154.533
C01720=1082.340,346.349,-93.838,176.273,26.889,154.532
C01721=1082.334,346.102,-93.804,176.270,26.884,154.531
C01722=1082.328,345.854,-93.769,176.267,26.879,154.530
C01723=1082.322,345.606,-93.735,176.263,26.874,154.529
C01724=1082.316,345.359,-93.699,176.260,26.869,154.529
C01725=1082.310,345.111,-93.665,176.257,26.864,154.528
C01726=1082.305,344.864,-93.631,176.255,26.859,154.527
C01727=1082.295,344.458,-93.574,176.249,26.850,154.526
C01728=1082.285,344.053,-93.517,176.244,26.842,154.524
C01729=1082.275,343.646,-93.460,176.239,26.834,154.523
C01730=1082.264,343.240,-93.404,176.234,26.826,154.522
C01731=1082.258,342.993,-93.370,176.231,26.821,154.521
C01732=1082.253,342.746,-93.335,176.227,26.816,154.520
C01733=1082.247,342.498,-93.301,176.224,26.811,154.519
C01734=1082.241,342.250,-93.267,176.221,26.806,154.518
C01735=1082.235,342.002,-93.232,176.218,26.801,154.518
C01736=1082.229,341.755,-93.198,176.215,26.796,154.517
C01737=1082.223,341.508,-93.164,176.211,26.791,154.516
C01738=1082.217,341.259,-93.129,176.208,26.786,154.515
C01739=1082.211,341.012,-93.095,176.205,26.782,154.514
C01740=1082.205,340.765,-93.061,176.202,26.777,154.514
C01741=1082.199,340.517,-93.026,176.199,26.772,154.513
C01742=1082.193,340.270,-92.992,176.195,26.767,154.512
C01743=1082.187,340.022,-92.958,176.192,26.762,154.511
C01744=1082.181,339.774,-92.924,176.189,26.757,154.510
C01745=1082.176,339.527,-92.889,176.186,26.752,154.510
C01746=1082.170,339.279,-92.855,176.183,26.747,154.509
C01747=1082.164,339.031,-92.822,176.180,26.743,154.508
C01748=1082.158,338.784,-92.787,176.176,26.737,154.507
C01749=1082.152,338.536,-92.753,176.174,26.733,154.506
C01750=1082.145,338.288,-92.719,176.171,26.728,154.506
C01751=1082.140,338.041,-92.685,176.168,26.723,154.505
C01752=1082.134,337.793,-92.652,176.164,26.719,154.504
C01753=1082.128,337.546,-92.618,176.162,26.714,154.503
C01754=1082.122,337.298,-92.583,176.158,26.709,154.503
C01755=1082.116,337.051,-92.549,176.155,26.704,154.502
C01756=1082.110,336.803,-92.516,176.152,26.699,154.501
C01757=1082.104,336.555,-92.481,176.149,26.694,154.500
C01758=1082.097,336.308,-92.448,176.146,26.690,154.500
C01759=1082.092,336.060,-92.415,176.143,26.685,154.499
C01760=1082.086,335.812,-92.380,176.140,26.681,154.498
C01761=1082.080,335.564,-92.347,176.136,26.675,154.497
C01762=1082.074,335.317,-92.313,176.133,26.671,154.497
C01763=1082.068,335.069,-92.279,176.130,26.666,154.496
C01764=1082.062,334.821,-92.245,176.127,26.662,154.495
C01765=1082.056,334.574,-92.211,176.124,26.657,154.494
C01766=1082.050,334.326,-92.178,176.121,26.652,154.494
C01767=1082.044,334.079,-92.144,176.118,26.648,154.493
C01768=1082.038,333.831,-92.111,176.115,26.643,154.492
C01769=1082.032,333.583,-92.077,176.112,26.639,154.491
C01770=1082.027,333.335,-92.043,176.108,26.633,154.491
C01771=1082.021,333.088,-92.009,176.105,26.629,154.490
C01772=1082.015,332.840,-91.976,176.102,26.624,154.489
C01773=1082.008,332.592,-91.943,176.099,26.619,154.488
C01774=1082.003,332.345,-91.909,176.096,26.615,154.488
C01775=1081.997,332.097,-91.876,176.093,26.610,154.487
C01776=1081.991,331.849,-91.841,176.090,26.606,154.486
C01777=1081.985,331.602,-91.809,176.087,26.601,154.486
C01778=1081.979,331.354,-91.775,176.084,26.596,154.485
C01779=1081.968,330.942,-91.720,176.079,26.589,154.484
C01780=1081.959,330.531,-91.664,176.073,26.581,154.483
C01781=1081.949,330.120,-91.609,176.068,26.574,154.481
C01782=1081.938,329.708,-91.554,176.064,26.567,154.480
C01783=1081.933,329.460,-91.521,176.061,26.562,154.480
C01784=1081.926,329.213,-91.487,176.058,26.557,154.479
C01785=1081.921,328.965,-91.454,176.054,26.553,154.478
C01786=1081.914,328.717,-91.421,176.051,26.548,154.477
C01787=1081.908,328.469,-91.388,176.048,26.544,154.477
C01788=1081.902,328.222,-91.355,176.045,26.539,154.476
C01789=1081.896,327.974,-91.322,176.042,26.535,154.475
C01790=1081.890,327.726,-91.289,176.038,26.531,154.475
C01791=1081.885,327.478,-91.256,176.035,26.526,154.474
C01792=1081.878,327.231,-91.223,176.033,26.522,154.473
C01793=1081.873,326.983,-91.189,176.029,26.517,154.473
C01794=1081.866,326.735,-91.157,176.026,26.513,154.472
C01795=1081.861,326.487,-91.123,176.023,26.509,154.471
C01796=1081.855,326.240,-91.091,176.020,26.504,154.471
C01797=1081.848,325.992,-91.058,176.017,26.499,154.470
C01798=1081.843,325.744,-91.025,176.014,26.495,154.469
C01799=1081.836,325.496,-90.992,176.011,26.491,154.469
C01800=1081.831,325.249,-90.958,176.008,26.486,154.468
